LIN {X 0,Y 178.486,Z 136.368,A -85,B 0,C 180,E1 -22471.803,E2 -22471.803} C_VEL
LIN {X 0,Y 178.51,Z 136.363,A -85,B 0,C 180,E1 -22476.815,E2 -22476.815} C_VEL
LIN {X 0,Y 178.649,Z 136.34,A -85,B 0,C 180,E1 -22481.657,E2 -22481.657} C_VEL
LIN {X 0,Y 178.666,Z 136.339,A -85,B 0,C 180,E1 -22486.349,E2 -22486.349} C_VEL
LIN {X 0,Y 178.957,Z 136.319,A -85,B 0,C 180,E1 -22490.962,E2 -22490.962} C_VEL
LIN {X 0,Y 179.152,Z 136.294,A -85,B 0,C 180,E1 -22497.752,E2 -22497.752} C_VEL
LIN {X 0,Y 179.369,Z 136.252,A -85,B 0,C 180,E1 -22500,E2 -22500} C_VEL
LIN {X 0,Y 178.86,Z 136.321,A -85,B 0,C 180,E1 -22504.508,E2 -22504.508} C_VEL
LIN {X 0,Y 178.907,Z 136.301,A -85,B 0,C 180,E1 -22509.041,E2 -22509.041} C_VEL
LIN {X 0,Y 178.659,Z 136.355,A -85,B 0,C 180,E1 -22513.653,E2 -22513.653} C_VEL
LIN {X 0,Y 178.654,Z 136.338,A -85,B 0,C 180,E1 -22519.245,E2 -22519.245} C_VEL
LIN {X 0,Y 178.535,Z 136.348,A -85,B 0,C 180,E1 -22525.125,E2 -22525.125} C_VEL
LIN {X 0,Y 178.522,Z 136.362,A -85,B 0,C 180,E1 -22529.994,E2 -22529.994} C_VEL
LIN {X 0,Y 178.484,Z 136.378,A -85,B 0,C 180,E1 -22534.22,E2 -22534.22} C_VEL
LIN {X 0,Y 178.434,Z 136.535,A -85,B 0,C 180,E1 -22539.429,E2 -22539.429} C_VEL
LIN {X 0,Y 179.248,Z 138.944,A -85,B 0,C 180,E1 -22539.944,E2 -22539.944} C_VEL
LIN {X 0,Y 181.215,Z 141.18,A -85,B 0,C 180,E1 -22540.917,E2 -22540.917} C_VEL
LIN {X 0,Y 182.206,Z 142.05,A -85,B 0,C 180,E1 -22541.375,E2 -22541.375} C_VEL
LIN {X 0,Y 184.192,Z 145.249,A -85,B 0,C 180,E1 -22542.353,E2 -22542.353} C_VEL
LIN {X 0,Y 185.848,Z 147.075,A -85,B 0,C 180,E1 -22543.088,E2 -22543.088} C_VEL
LIN {X 0,Y 188.488,Z 150.745,A -85,B 0,C 180,E1 -22544.254,E2 -22544.254} C_VEL
LIN {X 0,Y 195.166,Z 160.483,A -85,B 0,C 180,E1 -22546.984,E2 -22546.984} C_VEL
LIN {X 0,Y 201.382,Z 170.518,A -85,B 0,C 180,E1 -22549.304,E2 -22549.304} C_VEL
LIN {X 0,Y 207.113,Z 180.976,A -85,B 0,C 180,E1 -22551.304,E2 -22551.304} C_VEL
LIN {X 0,Y 212.528,Z 194.015,A -85,B 0,C 180,E1 -22553.179,E2 -22553.179} C_VEL
LIN {X 0,Y 208.581,Z 264.938,A -85,B 0,C 180,E1 -22555.422,E2 -22555.422} C_VEL
LIN {X 0,Y 207.1,Z 278.824,A -85,B 0,C 180,E1 -22556.169,E2 -22556.169} C_VEL
LIN {X 0,Y 204.905,Z 292.956,A -85,B 0,C 180,E1 -22557.303,E2 -22557.303} C_VEL
LIN {X 0,Y 201.992,Z 306.924,A -85,B 0,C 180,E1 -22558.832,E2 -22558.832} C_VEL
LIN {X 0,Y 198.824,Z 319.397,A -85,B 0,C 180,E1 -22560.63,E2 -22560.63} C_VEL
LIN {X 0,Y 195.579,Z 330.767,A -85,B 0,C 180,E1 -22562.732,E2 -22562.732} C_VEL
LIN {X 0,Y 192.154,Z 341.225,A -85,B 0,C 180,E1 -22565.127,E2 -22565.127} C_VEL
LIN {X 0,Y 188.423,Z 351.62,A -85,B 0,C 180,E1 -22568.1,E2 -22568.1} C_VEL
LIN {X 0,Y 185.325,Z 360.19,A -85,B 0,C 180,E1 -22571.196,E2 -22571.196} C_VEL
LIN {X 0,Y 182.454,Z 367.978,A -85,B 0,C 180,E1 -22574.699,E2 -22574.699} C_VEL
LIN {X 0,Y 179.719,Z 375.042,A -85,B 0,C 180,E1 -22578.725,E2 -22578.725} C_VEL
LIN {X 0,Y 177.688,Z 380.92,A -85,B 0,C 180,E1 -22583.186,E2 -22583.186} C_VEL
LIN {X 0,Y 176.565,Z 385.24,A -85,B 0,C 180,E1 -22587.719,E2 -22587.719} C_VEL
LIN {X 0,Y 176.02,Z 388.135,A -85,B 0,C 180,E1 -22592.289,E2 -22592.289} C_VEL
LIN {X 0,Y 175.937,Z 389.074,A -85,B 0,C 180,E1 -22594.583,E2 -22594.583} C_VEL
LIN {X 0,Y 175.912,Z 389.967,A -85,B 0,C 180,E1 -22599.196,E2 -22599.196} C_VEL
LIN {X 0,Y 176.481,Z 389.534,A -85,B 0,C 180,E1 -22603.824,E2 -22603.824} C_VEL
LIN {X 0,Y 177.992,Z 387.659,A -85,B 0,C 180,E1 -22608.622,E2 -22608.622} C_VEL
LIN {X 0,Y 180.078,Z 384.585,A -85,B 0,C 180,E1 -22612.972,E2 -22612.972} C_VEL
LIN {X 0,Y 183.234,Z 379.874,A -85,B 0,C 180,E1 -22617.405,E2 -22617.405} C_VEL
LIN {X 0,Y 186.251,Z 375.283,A -85,B 0,C 180,E1 -22620.625,E2 -22620.625} C_VEL
LIN {X 0,Y 190.461,Z 368.593,A -85,B 0,C 180,E1 -22624.245,E2 -22624.245} C_VEL
LIN {X 0,Y 195.256,Z 360.22,A -85,B 0,C 180,E1 -22627.727,E2 -22627.727} C_VEL
LIN {X 0,Y 199.905,Z 351.456,A -85,B 0,C 180,E1 -22630.572,E2 -22630.572} C_VEL
LIN {X 0,Y 204.196,Z 342.773,A -85,B 0,C 180,E1 -22632.825,E2 -22632.825} C_VEL
LIN {X 0,Y 209.112,Z 331.656,A -85,B 0,C 180,E1 -22635.107,E2 -22635.107} C_VEL
LIN {X 0,Y 213.096,Z 321.091,A -85,B 0,C 180,E1 -22636.861,E2 -22636.861} C_VEL
LIN {X 0,Y 217.194,Z 308.734,A -85,B 0,C 180,E1 -22638.442,E2 -22638.442} C_VEL
LIN {X 0,Y 220.596,Z 296.079,A -85,B 0,C 180,E1 -22639.697,E2 -22639.697} C_VEL
LIN {X 0,Y 223.426,Z 281.915,A -85,B 0,C 180,E1 -22640.76,E2 -22640.76} C_VEL
LIN {X 0,Y 225.438,Z 268.079,A -85,B 0,C 180,E1 -22641.453,E2 -22641.453} C_VEL
LIN {X 0,Y 227.196,Z 245.698,A -85,B 0,C 180,E1 -22642.138,E2 -22642.138} C_VEL
LIN {X 0,Y 229.57,Z 209.78,A -85,B 0,C 180,E1 -22643.147,E2 -22643.147} C_VEL
LIN {X 0,Y 223.747,Z 197.099,A -85,B 0,C 180,E1 -22645.613,E2 -22645.613} C_VEL
LIN {X 0,Y 219.607,Z 189.431,A -85,B 0,C 180,E1 -22647.466,E2 -22647.466} C_VEL
LIN {X 0,Y 213.902,Z 180.454,A -85,B 0,C 180,E1 -22650.201,E2 -22650.201} C_VEL
LIN {X 0,Y 208.778,Z 173.011,A -85,B 0,C 180,E1 -22652.947,E2 -22652.947} C_VEL
LIN {X 0,Y 205.032,Z 168.032,A -85,B 0,C 180,E1 -22655.171,E2 -22655.171} C_VEL
LIN {X 0,Y 202.022,Z 163.972,A -85,B 0,C 180,E1 -22657.155,E2 -22657.155} C_VEL
LIN {X 0,Y 199.176,Z 160.496,A -85,B 0,C 180,E1 -22659.202,E2 -22659.202} C_VEL
LIN {X 0,Y 198.282,Z 159.146,A -85,B 0,C 180,E1 -22659.917,E2 -22659.917} C_VEL
LIN {X 0,Y 195.65,Z 156.447,A -85,B 0,C 180,E1 -22662.073,E2 -22662.073} C_VEL
LIN {X 0,Y 194.186,Z 153.936,A -85,B 0,C 180,E1 -22663.508,E2 -22663.508} C_VEL
LIN {X 0,Y 191.565,Z 151.793,A -85,B 0,C 180,E1 -22666.136,E2 -22666.136} C_VEL
LIN {X 0,Y 189.782,Z 148.386,A -85,B 0,C 180,E1 -22668.518,E2 -22668.518} C_VEL
LIN {X 0,Y 186.239,Z 145.756,A -85,B 0,C 180,E1 -22674.315,E2 -22674.315} C_VEL
LIN {X 0,Y 185.281,Z 143.481,A -85,B 0,C 180,E1 -22677.418,E2 -22677.418} C_VEL
LIN {X 0,Y 185.143,Z 142.415,A -85,B 0,C 180,E1 -22678.368,E2 -22678.368} C_VEL
LIN {X 0,Y 185.004,Z 142.485,A -85,B 0,C 180,E1 -22686.817,E2 -22686.817} C_VEL
LIN {X 0,Y 186.711,Z 146.523,A -85,B 0,C 180,E1 -22692.499,E2 -22692.499} C_VEL
LIN {X 0,Y 189.834,Z 148.662,A -85,B 0,C 180,E1 -22697.311,E2 -22697.311} C_VEL
LIN {X 0,Y 191.307,Z 151.577,A -85,B 0,C 180,E1 -22699.307,E2 -22699.307} C_VEL
LIN {X 0,Y 193.883,Z 153.809,A -85,B 0,C 180,E1 -22701.951,E2 -22701.951} C_VEL
LIN {X 0,Y 194.461,Z 154.358,A -85,B 0,C 180,E1 -22702.494,E2 -22702.494} C_VEL
LIN {X 0,Y 196.476,Z 157.499,A -85,B 0,C 180,E1 -22704.38,E2 -22704.38} C_VEL
LIN {X 0,Y 198.823,Z 159.877,A -85,B 0,C 180,E1 -22706.239,E2 -22706.239} C_VEL
LIN {X 0,Y 201.386,Z 163.367,A -85,B 0,C 180,E1 -22708.148,E2 -22708.148} C_VEL
LIN {X 0,Y 203.327,Z 165.931,A -85,B 0,C 180,E1 -22709.473,E2 -22709.473} C_VEL
LIN {X 0,Y 207.068,Z 171.804,A -85,B 0,C 180,E1 -22711.87,E2 -22711.87} C_VEL
LIN {X 0,Y 209.974,Z 176.459,A -85,B 0,C 180,E1 -22713.567,E2 -22713.567} C_VEL
LIN {X 0,Y 214.704,Z 184.513,A -85,B 0,C 180,E1 -22716.1,E2 -22716.1} C_VEL
LIN {X 0,Y 220.915,Z 196.355,A -85,B 0,C 180,E1 -22719.107,E2 -22719.107} C_VEL
LIN {X 0,Y 226.829,Z 209.325,A -85,B 0,C 180,E1 -22721.726,E2 -22721.726} C_VEL
LIN {X 0,Y 229.29,Z 215.482,A -85,B 0,C 180,E1 -22722.771,E2 -22722.771} C_VEL
LIN {X 0,Y 226.765,Z 253.212,A -85,B 0,C 180,E1 -22723.821,E2 -22723.821} C_VEL
LIN {X 0,Y 225.889,Z 259.067,A -85,B 0,C 180,E1 -22723.837,E2 -22723.837} C_VEL
LIN {X 0,Y 220.831,Z 276.116,A -85,B 0,C 180,E1 -22723.343,E2 -22723.343} C_VEL
LIN {X 0,Y 219.402,Z 281.85,A -85,B 0,C 180,E1 -22723.411,E2 -22723.411} C_VEL
LIN {X 0,Y 219.081,Z 283.768,A -85,B 0,C 180,E1 -22723.5,E2 -22723.5} C_VEL
LIN {X 0,Y 216.297,Z 297.815,A -85,B 0,C 180,E1 -22724.37,E2 -22724.37} C_VEL
LIN {X 0,Y 212.928,Z 310.546,A -85,B 0,C 180,E1 -22725.461,E2 -22725.461} C_VEL
LIN {X 0,Y 208.683,Z 323.745,A -85,B 0,C 180,E1 -22727.001,E2 -22727.001} C_VEL
LIN {X 0,Y 204.032,Z 335.665,A -85,B 0,C 180,E1 -22728.794,E2 -22728.794} C_VEL
LIN {X 0,Y 198.988,Z 347.089,A -85,B 0,C 180,E1 -22731.032,E2 -22731.032} C_VEL
LIN {X 0,Y 193.433,Z 358.123,A -85,B 0,C 180,E1 -22733.813,E2 -22733.813} C_VEL
LIN {X 0,Y 188.464,Z 366.89,A -85,B 0,C 180,E1 -22736.63,E2 -22736.63} C_VEL
LIN {X 0,Y 183.38,Z 375.311,A -85,B 0,C 180,E1 -22740.117,E2 -22740.117} C_VEL
LIN {X 0,Y 179.533,Z 381.206,A -85,B 0,C 180,E1 -22743.245,E2 -22743.245} C_VEL
LIN {X 0,Y 176.298,Z 386.092,A -85,B 0,C 180,E1 -22746.506,E2 -22746.506} C_VEL
LIN {X 0,Y 173.054,Z 391.158,A -85,B 0,C 180,E1 -22751.041,E2 -22751.041} C_VEL
LIN {X 0,Y 170.616,Z 394.743,A -85,B 0,C 180,E1 -22755.691,E2 -22755.691} C_VEL
LIN {X 0,Y 169.324,Z 396.953,A -85,B 0,C 180,E1 -22760.443,E2 -22760.443} C_VEL
LIN {X 0,Y 168.858,Z 397.835,A -85,B 0,C 180,E1 -22765.225,E2 -22765.225} C_VEL
LIN {X 0,Y 168.943,Z 397.392,A -85,B 0,C 180,E1 -22770,E2 -22770} C_VEL
LIN {X 0,Y 168.833,Z 396.62,A -85,B 0,C 180,E1 -22772.506,E2 -22772.506} C_VEL
LIN {X 0,Y 168.962,Z 394.168,A -85,B 0,C 180,E1 -22777.168,E2 -22777.168} C_VEL
LIN {X 0,Y 169.478,Z 391.316,A -85,B 0,C 180,E1 -22780.754,E2 -22780.754} C_VEL
LIN {X 0,Y 170.853,Z 386.202,A -85,B 0,C 180,E1 -22785.508,E2 -22785.508} C_VEL
LIN {X 0,Y 172.563,Z 381.246,A -85,B 0,C 180,E1 -22789.015,E2 -22789.015} C_VEL
LIN {X 0,Y 175.147,Z 374.083,A -85,B 0,C 180,E1 -22793.045,E2 -22793.045} C_VEL
LIN {X 0,Y 178.555,Z 365.268,A -85,B 0,C 180,E1 -22796.913,E2 -22796.913} C_VEL
LIN {X 0,Y 182.099,Z 356.008,A -85,B 0,C 180,E1 -22800.114,E2 -22800.114} C_VEL
LIN {X 0,Y 185.95,Z 345.785,A -85,B 0,C 180,E1 -22802.908,E2 -22802.908} C_VEL
LIN {X 0,Y 189.809,Z 334.101,A -85,B 0,C 180,E1 -22805.454,E2 -22805.454} C_VEL
LIN {X 0,Y 193.369,Z 322.05,A -85,B 0,C 180,E1 -22807.501,E2 -22807.501} C_VEL
LIN {X 0,Y 196.679,Z 309.03,A -85,B 0,C 180,E1 -22809.2,E2 -22809.2} C_VEL
LIN {X 0,Y 199.46,Z 295.554,A -85,B 0,C 180,E1 -22810.514,E2 -22810.514} C_VEL
LIN {X 0,Y 201.683,Z 280.974,A -85,B 0,C 180,E1 -22811.525,E2 -22811.525} C_VEL
LIN {X 0,Y 203.143,Z 266.315,A -85,B 0,C 180,E1 -22812.156,E2 -22812.156} C_VEL
LIN {X 0,Y 206.817,Z 201.907,A -85,B 0,C 180,E1 -22814.192,E2 -22814.192} C_VEL
LIN {X 0,Y 201.234,Z 187.244,A -85,B 0,C 180,E1 -22816.303,E2 -22816.303} C_VEL
LIN {X 0,Y 195.797,Z 175.404,A -85,B 0,C 180,E1 -22818.428,E2 -22818.428} C_VEL
LIN {X 0,Y 189.888,Z 163.919,A -85,B 0,C 180,E1 -22820.901,E2 -22820.901} C_VEL
LIN {X 0,Y 186.31,Z 158.007,A -85,B 0,C 180,E1 -22822.476,E2 -22822.476} C_VEL
LIN {X 0,Y 181.962,Z 151.818,A -85,B 0,C 180,E1 -22824.488,E2 -22824.488} C_VEL
LIN {X 0,Y 179.388,Z 148.301,A -85,B 0,C 180,E1 -22825.76,E2 -22825.76} C_VEL
LIN {X 0,Y 176.29,Z 144.63,A -85,B 0,C 180,E1 -22827.355,E2 -22827.355} C_VEL
LIN {X 0,Y 175.102,Z 142.606,A -85,B 0,C 180,E1 -22828.042,E2 -22828.042} C_VEL
LIN {X 0,Y 172.77,Z 140.563,A -85,B 0,C 180,E1 -22829.313,E2 -22829.313} C_VEL
LIN {X 0,Y 171.595,Z 137.936,A -85,B 0,C 180,E1 -22830.104,E2 -22830.104} C_VEL
LIN {X 0,Y 171.472,Z 137.24,A -85,B 0,C 180,E1 -22830.31,E2 -22830.31} C_VEL
LIN {X 0,Y 171.457,Z 137.238,A -85,B 0,C 180,E1 -22835.802,E2 -22835.802} C_VEL
LIN {X 0,Y 171.578,Z 137.22,A -85,B 0,C 180,E1 -22840.872,E2 -22840.872} C_VEL
LIN {X 0,Y 171.593,Z 137.225,A -85,B 0,C 180,E1 -22845.775,E2 -22845.775} C_VEL
LIN {X 0,Y 171.886,Z 137.199,A -85,B 0,C 180,E1 -22850.587,E2 -22850.587} C_VEL
LIN {X 0,Y 171.818,Z 137.189,A -85,B 0,C 180,E1 -22855.308,E2 -22855.308} C_VEL
LIN {X 0,Y 172.332,Z 137.127,A -85,B 0,C 180,E1 -22860,E2 -22860} C_VEL
LIN {X 0,Y 171.809,Z 137.201,A -85,B 0,C 180,E1 -22864.693,E2 -22864.693} C_VEL
LIN {X 0,Y 171.844,Z 137.177,A -85,B 0,C 180,E1 -22869.416,E2 -22869.416} C_VEL
LIN {X 0,Y 171.58,Z 137.237,A -85,B 0,C 180,E1 -22874.227,E2 -22874.227} C_VEL
LIN {X 0,Y 171.575,Z 137.222,A -85,B 0,C 180,E1 -22879.591,E2 -22879.591} C_VEL
LIN {X 0,Y 171.469,Z 137.228,A -85,B 0,C 180,E1 -22885.617,E2 -22885.617} C_VEL
LIN {X 0,Y 171.441,Z 137.239,A -85,B 0,C 180,E1 -22890.587,E2 -22890.587} C_VEL
LIN {X 0,Y 171.393,Z 137.302,A -85,B 0,C 180,E1 -22896.119,E2 -22896.119} C_VEL
LIN {X 0,Y 172.221,Z 139.853,A -85,B 0,C 180,E1 -22896.734,E2 -22896.734} C_VEL
LIN {X 0,Y 174.207,Z 142.08,A -85,B 0,C 180,E1 -22897.872,E2 -22897.872} C_VEL
LIN {X 0,Y 175.392,Z 143.049,A -85,B 0,C 180,E1 -22898.499,E2 -22898.499} C_VEL
LIN {X 0,Y 177.484,Z 146.372,A -85,B 0,C 180,E1 -22899.671,E2 -22899.671} C_VEL
LIN {X 0,Y 179.247,Z 148.253,A -85,B 0,C 180,E1 -22900.553,E2 -22900.553} C_VEL
LIN {X 0,Y 181.957,Z 151.964,A -85,B 0,C 180,E1 -22901.895,E2 -22901.895} C_VEL
LIN {X 0,Y 186.526,Z 158.471,A -85,B 0,C 180,E1 -22904.004,E2 -22904.004} C_VEL
LIN {X 0,Y 191.824,Z 166.326,A -85,B 0,C 180,E1 -22906.24,E2 -22906.24} C_VEL
LIN {X 0,Y 198.165,Z 176.886,A -85,B 0,C 180,E1 -22908.714,E2 -22908.714} C_VEL
LIN {X 0,Y 202.96,Z 185.998,A -85,B 0,C 180,E1 -22910.473,E2 -22910.473} C_VEL
LIN {X 0,Y 207.061,Z 196.134,A -85,B 0,C 180,E1 -22911.982,E2 -22911.982} C_VEL
LIN {X 0,Y 203.045,Z 264.915,A -85,B 0,C 180,E1 -22914.185,E2 -22914.185} C_VEL
LIN {X 0,Y 201.518,Z 278.875,A -85,B 0,C 180,E1 -22914.946,E2 -22914.946} C_VEL
LIN {X 0,Y 199.231,Z 293.039,A -85,B 0,C 180,E1 -22916.097,E2 -22916.097} C_VEL
LIN {X 0,Y 196.41,Z 306.148,A -85,B 0,C 180,E1 -22917.539,E2 -22917.539} C_VEL
LIN {X 0,Y 193.091,Z 318.804,A -85,B 0,C 180,E1 -22919.366,E2 -22919.366} C_VEL
LIN {X 0,Y 189.707,Z 330.306,A -85,B 0,C 180,E1 -22921.512,E2 -22921.512} C_VEL
LIN {X 0,Y 185.758,Z 341.839,A -85,B 0,C 180,E1 -22924.209,E2 -22924.209} C_VEL
LIN {X 0,Y 181.879,Z 352.16,A -85,B 0,C 180,E1 -22927.269,E2 -22927.269} C_VEL
LIN {X 0,Y 178.643,Z 360.666,A -85,B 0,C 180,E1 -22930.464,E2 -22930.464} C_VEL
LIN {X 0,Y 175.825,Z 367.743,A -85,B 0,C 180,E1 -22933.752,E2 -22933.752} C_VEL
LIN {X 0,Y 173.513,Z 373.633,A -85,B 0,C 180,E1 -22937.128,E2 -22937.128} C_VEL
LIN {X 0,Y 171.175,Z 379.925,A -85,B 0,C 180,E1 -22941.738,E2 -22941.738} C_VEL
LIN {X 0,Y 169.997,Z 383.551,A -85,B 0,C 180,E1 -22945.258,E2 -22945.258} C_VEL
LIN {X 0,Y 169.119,Z 387.107,A -85,B 0,C 180,E1 -22950,E2 -22950} C_VEL
LIN {X 0,Y 168.912,Z 388.672,A -85,B 0,C 180,E1 -22953.043,E2 -22953.043} C_VEL
LIN {X 0,Y 168.774,Z 389.877,A -85,B 0,C 180,E1 -22957.177,E2 -22957.177} C_VEL
LIN {X 0,Y 169.03,Z 390.073,A -85,B 0,C 180,E1 -22961.999,E2 -22961.999} C_VEL
LIN {X 0,Y 170.17,Z 388.934,A -85,B 0,C 180,E1 -22966.804,E2 -22966.804} C_VEL
LIN {X 0,Y 172.11,Z 386.428,A -85,B 0,C 180,E1 -22971.562,E2 -22971.562} C_VEL
LIN {X 0,Y 175.033,Z 382.448,A -85,B 0,C 180,E1 -22976.211,E2 -22976.211} C_VEL
LIN {X 0,Y 178.908,Z 376.877,A -85,B 0,C 180,E1 -22980.709,E2 -22980.709} C_VEL
LIN {X 0,Y 183.174,Z 370.555,A -85,B 0,C 180,E1 -22984.467,E2 -22984.467} C_VEL
LIN {X 0,Y 187.755,Z 363.199,A -85,B 0,C 180,E1 -22987.844,E2 -22987.844} C_VEL
LIN {X 0,Y 192.785,Z 354.366,A -85,B 0,C 180,E1 -22991.01,E2 -22991.01} C_VEL
LIN {X 0,Y 198.038,Z 344.351,A -85,B 0,C 180,E1 -22993.79,E2 -22993.79} C_VEL
LIN {X 0,Y 202.947,Z 334.007,A -85,B 0,C 180,E1 -22996.022,E2 -22996.022} C_VEL
LIN {X 0,Y 207.194,Z 323.327,A -85,B 0,C 180,E1 -22997.902,E2 -22997.902} C_VEL
LIN {X 0,Y 211.493,Z 311.505,A -85,B 0,C 180,E1 -22999.477,E2 -22999.477} C_VEL
LIN {X 0,Y 214.919,Z 299.537,A -85,B 0,C 180,E1 -23000.769,E2 -23000.769} C_VEL
LIN {X 0,Y 218.012,Z 285.863,A -85,B 0,C 180,E1 -23001.885,E2 -23001.885} C_VEL
LIN {X 0,Y 220.37,Z 271.605,A -85,B 0,C 180,E1 -23002.688,E2 -23002.688} C_VEL
LIN {X 0,Y 221.867,Z 256.171,A -85,B 0,C 180,E1 -23003.228,E2 -23003.228} C_VEL
LIN {X 0,Y 224.935,Z 212.537,A -85,B 0,C 180,E1 -23004.439,E2 -23004.439} C_VEL
LIN {X 0,Y 219.404,Z 200.419,A -85,B 0,C 180,E1 -23006.937,E2 -23006.937} C_VEL
LIN {X 0,Y 215.998,Z 194.049,A -85,B 0,C 180,E1 -23008.559,E2 -23008.559} C_VEL
LIN {X 0,Y 210.252,Z 184.968,A -85,B 0,C 180,E1 -23011.485,E2 -23011.485} C_VEL
LIN {X 0,Y 205.74,Z 178.356,A -85,B 0,C 180,E1 -23014.061,E2 -23014.061} C_VEL
LIN {X 0,Y 202.638,Z 174.042,A -85,B 0,C 180,E1 -23016.016,E2 -23016.016} C_VEL
LIN {X 0,Y 199.776,Z 170.125,A -85,B 0,C 180,E1 -23018,E2 -23018} C_VEL
LIN {X 0,Y 197.006,Z 166.47,A -85,B 0,C 180,E1 -23020.122,E2 -23020.122} C_VEL
LIN {X 0,Y 196.04,Z 165.384,A -85,B 0,C 180,E1 -23020.905,E2 -23020.905} C_VEL
LIN {X 0,Y 193.487,Z 162.209,A -85,B 0,C 180,E1 -23023.192,E2 -23023.192} C_VEL
LIN {X 0,Y 192.499,Z 160.599,A -85,B 0,C 180,E1 -23024.21,E2 -23024.21} C_VEL
LIN {X 0,Y 189.879,Z 158.11,A -85,B 0,C 180,E1 -23027.032,E2 -23027.032} C_VEL
LIN {X 0,Y 188.318,Z 155.191,A -85,B 0,C 180,E1 -23029.245,E2 -23029.245} C_VEL
LIN {X 0,Y 184.947,Z 152.273,A -85,B 0,C 180,E1 -23035.368,E2 -23035.368} C_VEL
LIN {X 0,Y 184.246,Z 149.993,A -85,B 0,C 180,E1 -23038.224,E2 -23038.224} C_VEL
LIN {X 0,Y 184.15,Z 149.427,A -85,B 0,C 180,E1 -23038.906,E2 -23038.906} C_VEL
LIN {X 0,Y 184.083,Z 149.537,A -85,B 0,C 180,E1 -23046.576,E2 -23046.576} C_VEL
LIN {X 0,Y 185.721,Z 153.53,A -85,B 0,C 180,E1 -23052.287,E2 -23052.287} C_VEL
LIN {X 0,Y 188.478,Z 155.492,A -85,B 0,C 180,E1 -23056.727,E2 -23056.727} C_VEL
LIN {X 0,Y 190.072,Z 158.501,A -85,B 0,C 180,E1 -23058.951,E2 -23058.951} C_VEL
LIN {X 0,Y 192.868,Z 161.11,A -85,B 0,C 180,E1 -23061.896,E2 -23061.896} C_VEL
LIN {X 0,Y 195.276,Z 164.638,A -85,B 0,C 180,E1 -23064.191,E2 -23064.191} C_VEL
LIN {X 0,Y 197.012,Z 166.46,A -85,B 0,C 180,E1 -23065.61,E2 -23065.61} C_VEL
LIN {X 0,Y 200.96,Z 171.847,A -85,B 0,C 180,E1 -23068.581,E2 -23068.581} C_VEL
LIN {X 0,Y 205.164,Z 178.66,A -85,B 0,C 180,E1 -23071.397,E2 -23071.397} C_VEL
LIN {X 0,Y 209.109,Z 185.297,A -85,B 0,C 180,E1 -23073.75,E2 -23073.75} C_VEL
LIN {X 0,Y 214.505,Z 195.407,A -85,B 0,C 180,E1 -23076.665,E2 -23076.665} C_VEL
LIN {X 0,Y 219.297,Z 205.378,A -85,B 0,C 180,E1 -23079.022,E2 -23079.022} C_VEL
LIN {X 0,Y 223.957,Z 216.249,A -85,B 0,C 180,E1 -23081.163,E2 -23081.163} C_VEL
LIN {X 0,Y 224.59,Z 217.837,A -85,B 0,C 180,E1 -23081.445,E2 -23081.445} C_VEL
LIN {X 0,Y 220.71,Z 272.075,A -85,B 0,C 180,E1 -23082.997,E2 -23082.997} C_VEL
LIN {X 0,Y 219.081,Z 283.768,A -85,B 0,C 180,E1 -23083.5,E2 -23083.5} C_VEL
LIN {X 0,Y 217.68,Z 289.476,A -85,B 0,C 180,E1 -23083.681,E2 -23083.681} C_VEL
LIN {X 0,Y 213.779,Z 298.62,A -85,B 0,C 180,E1 -23083.711,E2 -23083.711} C_VEL
LIN {X 0,Y 209.463,Z 307.524,A -85,B 0,C 180,E1 -23083.88,E2 -23083.88} C_VEL
LIN {X 0,Y 207.419,Z 312.852,A -85,B 0,C 180,E1 -23084.29,E2 -23084.29} C_VEL
LIN {X 0,Y 202.99,Z 325.564,A -85,B 0,C 180,E1 -23085.831,E2 -23085.831} C_VEL
LIN {X 0,Y 198.232,Z 337.132,A -85,B 0,C 180,E1 -23087.653,E2 -23087.653} C_VEL
LIN {X 0,Y 192.771,Z 348.823,A -85,B 0,C 180,E1 -23090.054,E2 -23090.054} C_VEL
LIN {X 0,Y 187.755,Z 358.279,A -85,B 0,C 180,E1 -23092.535,E2 -23092.535} C_VEL
LIN {X 0,Y 182.55,Z 366.993,A -85,B 0,C 180,E1 -23095.399,E2 -23095.399} C_VEL
LIN {X 0,Y 177.222,Z 375.368,A -85,B 0,C 180,E1 -23098.967,E2 -23098.967} C_VEL
LIN {X 0,Y 173.203,Z 381.22,A -85,B 0,C 180,E1 -23102.184,E2 -23102.184} C_VEL
LIN {X 0,Y 169.592,Z 386.311,A -85,B 0,C 180,E1 -23105.74,E2 -23105.74} C_VEL
LIN {X 0,Y 166.295,Z 391.098,A -85,B 0,C 180,E1 -23110.239,E2 -23110.239} C_VEL
LIN {X 0,Y 163.7,Z 394.649,A -85,B 0,C 180,E1 -23115.072,E2 -23115.072} C_VEL
LIN {X 0,Y 162.311,Z 396.828,A -85,B 0,C 180,E1 -23120.026,E2 -23120.026} C_VEL
LIN {X 0,Y 161.76,Z 397.679,A -85,B 0,C 180,E1 -23125.015,E2 -23125.015} C_VEL
LIN {X 0,Y 161.761,Z 397.591,A -85,B 0,C 180,E1 -23127.817,E2 -23127.817} C_VEL
LIN {X 0,Y 161.842,Z 397.206,A -85,B 0,C 180,E1 -23130,E2 -23130} C_VEL
LIN {X 0,Y 161.756,Z 396.46,A -85,B 0,C 180,E1 -23132.49,E2 -23132.49} C_VEL
LIN {X 0,Y 161.905,Z 393.932,A -85,B 0,C 180,E1 -23137.482,E2 -23137.482} C_VEL
LIN {X 0,Y 162.742,Z 389.93,A -85,B 0,C 180,E1 -23142.469,E2 -23142.469} C_VEL
LIN {X 0,Y 164.543,Z 384.342,A -85,B 0,C 180,E1 -23147.396,E2 -23147.396} C_VEL
LIN {X 0,Y 166.893,Z 378.022,A -85,B 0,C 180,E1 -23151.621,E2 -23151.621} C_VEL
LIN {X 0,Y 170.036,Z 370.14,A -85,B 0,C 180,E1 -23155.721,E2 -23155.721} C_VEL
LIN {X 0,Y 173.395,Z 361.9,A -85,B 0,C 180,E1 -23159.103,E2 -23159.103} C_VEL
LIN {X 0,Y 177.421,Z 351.972,A -85,B 0,C 180,E1 -23162.327,E2 -23162.327} C_VEL
LIN {X 0,Y 181.523,Z 340.924,A -85,B 0,C 180,E1 -23165.163,E2 -23165.163} C_VEL
LIN {X 0,Y 185.554,Z 328.619,A -85,B 0,C 180,E1 -23167.643,E2 -23167.643} C_VEL
LIN {X 0,Y 189.098,Z 316.411,A -85,B 0,C 180,E1 -23169.528,E2 -23169.528} C_VEL
LIN {X 0,Y 192.391,Z 302.85,A -85,B 0,C 180,E1 -23171.112,E2 -23171.112} C_VEL
LIN {X 0,Y 195.077,Z 288.65,A -85,B 0,C 180,E1 -23172.318,E2 -23172.318} C_VEL
LIN {X 0,Y 197.02,Z 273.931,A -85,B 0,C 180,E1 -23173.163,E2 -23173.163} C_VEL
LIN {X 0,Y 198.847,Z 247.466,A -85,B 0,C 180,E1 -23174.059,E2 -23174.059} C_VEL
LIN {X 0,Y 201.431,Z 203.981,A -85,B 0,C 180,E1 -23175.451,E2 -23175.451} C_VEL
LIN {X 0,Y 195.716,Z 188.866,A -85,B 0,C 180,E1 -23177.765,E2 -23177.765} C_VEL
LIN {X 0,Y 189.867,Z 176.201,A -85,B 0,C 180,E1 -23180.233,E2 -23180.233} C_VEL
LIN {X 0,Y 183.905,Z 164.91,A -85,B 0,C 180,E1 -23182.948,E2 -23182.948} C_VEL
LIN {X 0,Y 178.64,Z 157.349,A -85,B 0,C 180,E1 -23185.486,E2 -23185.486} C_VEL
LIN {X 0,Y 175.577,Z 153.226,A -85,B 0,C 180,E1 -23187.088,E2 -23187.088} C_VEL
LIN {X 0,Y 173,Z 149.834,A -85,B 0,C 180,E1 -23188.527,E2 -23188.527} C_VEL
LIN {X 0,Y 172.172,Z 148.661,A -85,B 0,C 180,E1 -23189.016,E2 -23189.016} C_VEL
LIN {X 0,Y 169.628,Z 145.845,A -85,B 0,C 180,E1 -23190.528,E2 -23190.528} C_VEL
LIN {X 0,Y 168.455,Z 143.707,A -85,B 0,C 180,E1 -23191.329,E2 -23191.329} C_VEL
LIN {X 0,Y 166.023,Z 141.89,A -85,B 0,C 180,E1 -23192.865,E2 -23192.865} C_VEL
LIN {X 0,Y 164.703,Z 139.463,A -85,B 0,C 180,E1 -23193.875,E2 -23193.875} C_VEL
LIN {X 0,Y 164.433,Z 138.119,A -85,B 0,C 180,E1 -23194.259,E2 -23194.259} C_VEL
LIN {X 0,Y 164.484,Z 138.108,A -85,B 0,C 180,E1 -23200.051,E2 -23200.051} C_VEL
LIN {X 0,Y 164.542,Z 138.11,A -85,B 0,C 180,E1 -23205.151,E2 -23205.151} C_VEL
LIN {X 0,Y 164.801,Z 138.08,A -85,B 0,C 180,E1 -23210.179,E2 -23210.179} C_VEL
LIN {X 0,Y 164.848,Z 138.062,A -85,B 0,C 180,E1 -23212.652,E2 -23212.652} C_VEL
LIN {X 0,Y 165.048,Z 138.051,A -85,B 0,C 180,E1 -23217.56,E2 -23217.56} C_VEL
LIN {X 0,Y 165.294,Z 138.002,A -85,B 0,C 180,E1 -23220,E2 -23220} C_VEL
LIN {X 0,Y 164.757,Z 138.08,A -85,B 0,C 180,E1 -23224.894,E2 -23224.894} C_VEL
LIN {X 0,Y 164.825,Z 138.07,A -85,B 0,C 180,E1 -23227.35,E2 -23227.35} C_VEL
LIN {X 0,Y 164.702,Z 138.068,A -85,B 0,C 180,E1 -23231.061,E2 -23231.061} C_VEL
LIN {X 0,Y 164.503,Z 138.092,A -85,B 0,C 180,E1 -23237.402,E2 -23237.402} C_VEL
LIN {X 0,Y 164.52,Z 138.105,A -85,B 0,C 180,E1 -23239.984,E2 -23239.984} C_VEL
LIN {X 0,Y 164.394,Z 138.111,A -85,B 0,C 180,E1 -23246.135,E2 -23246.135} C_VEL
LIN {X 0,Y 164.394,Z 138.247,A -85,B 0,C 180,E1 -23252.199,E2 -23252.199} C_VEL
LIN {X 0,Y 165.252,Z 140.842,A -85,B 0,C 180,E1 -23252.958,E2 -23252.958} C_VEL
LIN {X 0,Y 167.27,Z 143.042,A -85,B 0,C 180,E1 -23254.331,E2 -23254.331} C_VEL
LIN {X 0,Y 168.599,Z 143.93,A -85,B 0,C 180,E1 -23255.144,E2 -23255.144} C_VEL
LIN {X 0,Y 170.318,Z 146.916,A -85,B 0,C 180,E1 -23256.291,E2 -23256.291} C_VEL
LIN {X 0,Y 172.64,Z 149.319,A -85,B 0,C 180,E1 -23257.636,E2 -23257.636} C_VEL
LIN {X 0,Y 175.288,Z 152.993,A -85,B 0,C 180,E1 -23259.14,E2 -23259.14} C_VEL
LIN {X 0,Y 176.681,Z 154.864,A -85,B 0,C 180,E1 -23259.887,E2 -23259.887} C_VEL
LIN {X 0,Y 180.01,Z 159.435,A -85,B 0,C 180,E1 -23261.585,E2 -23261.585} C_VEL
LIN {X 0,Y 185.561,Z 167.501,A -85,B 0,C 180,E1 -23264.182,E2 -23264.182} C_VEL
LIN {X 0,Y 191.821,Z 177.649,A -85,B 0,C 180,E1 -23266.848,E2 -23266.848} C_VEL
LIN {X 0,Y 198.206,Z 189.59,A -85,B 0,C 180,E1 -23269.358,E2 -23269.358} C_VEL
LIN {X 0,Y 201.692,Z 198.33,A -85,B 0,C 180,E1 -23270.725,E2 -23270.725} C_VEL
LIN {X 0,Y 197.456,Z 266.085,A -85,B 0,C 180,E1 -23272.926,E2 -23272.926} C_VEL
LIN {X 0,Y 195.796,Z 280.424,A -85,B 0,C 180,E1 -23273.763,E2 -23273.763} C_VEL
LIN {X 0,Y 193.431,Z 294.228,A -85,B 0,C 180,E1 -23274.934,E2 -23274.934} C_VEL
LIN {X 0,Y 190.49,Z 307.117,A -85,B 0,C 180,E1 -23276.399,E2 -23276.399} C_VEL
LIN {X 0,Y 187.056,Z 319.617,A -85,B 0,C 180,E1 -23278.265,E2 -23278.265} C_VEL
LIN {X 0,Y 183.521,Z 331.006,A -85,B 0,C 180,E1 -23280.459,E2 -23280.459} C_VEL
LIN {X 0,Y 179.42,Z 342.45,A -85,B 0,C 180,E1 -23283.227,E2 -23283.227} C_VEL
LIN {X 0,Y 175.388,Z 352.686,A -85,B 0,C 180,E1 -23286.378,E2 -23286.378} C_VEL
LIN {X 0,Y 171.995,Z 361.135,A -85,B 0,C 180,E1 -23289.677,E2 -23289.677} C_VEL
LIN {X 0,Y 168.6,Z 369.22,A -85,B 0,C 180,E1 -23293.659,E2 -23293.659} C_VEL
LIN {X 0,Y 165.852,Z 375.741,A -85,B 0,C 180,E1 -23297.768,E2 -23297.768} C_VEL
LIN {X 0,Y 163.639,Z 381.533,A -85,B 0,C 180,E1 -23302.598,E2 -23302.598} C_VEL
LIN {X 0,Y 162.395,Z 385.772,A -85,B 0,C 180,E1 -23307.52,E2 -23307.52} C_VEL
LIN {X 0,Y 161.835,Z 388.717,A -85,B 0,C 180,E1 -23312.769,E2 -23312.769} C_VEL
LIN {X 0,Y 161.679,Z 390.069,A -85,B 0,C 180,E1 -23317.493,E2 -23317.493} C_VEL
LIN {X 0,Y 162.001,Z 390.229,A -85,B 0,C 180,E1 -23322.528,E2 -23322.528} C_VEL
LIN {X 0,Y 163.286,Z 389.051,A -85,B 0,C 180,E1 -23327.535,E2 -23327.535} C_VEL
LIN {X 0,Y 165.404,Z 386.495,A -85,B 0,C 180,E1 -23332.483,E2 -23332.483} C_VEL
LIN {X 0,Y 168.553,Z 382.468,A -85,B 0,C 180,E1 -23337.301,E2 -23337.301} C_VEL
LIN {X 0,Y 172.736,Z 376.854,A -85,B 0,C 180,E1 -23341.933,E2 -23341.933} C_VEL
LIN {X 0,Y 177.244,Z 370.485,A -85,B 0,C 180,E1 -23345.794,E2 -23345.794} C_VEL
LIN {X 0,Y 182.367,Z 362.62,A -85,B 0,C 180,E1 -23349.434,E2 -23349.434} C_VEL
LIN {X 0,Y 187.393,Z 354.185,A -85,B 0,C 180,E1 -23352.46,E2 -23352.46} C_VEL
LIN {X 0,Y 192.911,Z 344.101,A -85,B 0,C 180,E1 -23355.269,E2 -23355.269} C_VEL
LIN {X 0,Y 198.362,Z 332.855,A -85,B 0,C 180,E1 -23357.687,E2 -23357.687} C_VEL
LIN {X 0,Y 203.012,Z 321.536,A -85,B 0,C 180,E1 -23359.607,E2 -23359.607} C_VEL
LIN {X 0,Y 207.394,Z 309.207,A -85,B 0,C 180,E1 -23361.206,E2 -23361.206} C_VEL
LIN {X 0,Y 211.035,Z 296.595,A -85,B 0,C 180,E1 -23362.469,E2 -23362.469} C_VEL
LIN {X 0,Y 214.047,Z 282.4,A -85,B 0,C 180,E1 -23363.557,E2 -23363.557} C_VEL
LIN {X 0,Y 216.292,Z 268.152,A -85,B 0,C 180,E1 -23364.259,E2 -23364.259} C_VEL
LIN {X 0,Y 218.211,Z 245.091,A -85,B 0,C 180,E1 -23364.967,E2 -23364.967} C_VEL
LIN {X 0,Y 220.404,Z 215.313,A -85,B 0,C 180,E1 -23365.79,E2 -23365.79} C_VEL
LIN {X 0,Y 215.532,Z 204.477,A -85,B 0,C 180,E1 -23368.14,E2 -23368.14} C_VEL
LIN {X 0,Y 212.34,Z 198.482,A -85,B 0,C 180,E1 -23369.754,E2 -23369.754} C_VEL
LIN {X 0,Y 206.325,Z 188.743,A -85,B 0,C 180,E1 -23373.051,E2 -23373.051} C_VEL
LIN {X 0,Y 200.866,Z 180.758,A -85,B 0,C 180,E1 -23376.494,E2 -23376.494} C_VEL
LIN {X 0,Y 197.7,Z 176.45,A -85,B 0,C 180,E1 -23378.767,E2 -23378.767} C_VEL
LIN {X 0,Y 194.518,Z 172.113,A -85,B 0,C 180,E1 -23381.367,E2 -23381.367} C_VEL
LIN {X 0,Y 191.881,Z 168.834,A -85,B 0,C 180,E1 -23383.816,E2 -23383.816} C_VEL
LIN {X 0,Y 191.098,Z 167.399,A -85,B 0,C 180,E1 -23384.672,E2 -23384.672} C_VEL
LIN {X 0,Y 188.508,Z 164.832,A -85,B 0,C 180,E1 -23387.587,E2 -23387.587} C_VEL
LIN {X 0,Y 187.059,Z 162.086,A -85,B 0,C 180,E1 -23389.74,E2 -23389.74} C_VEL
LIN {X 0,Y 183.919,Z 159.168,A -85,B 0,C 180,E1 -23395.788,E2 -23395.788} C_VEL
LIN {X 0,Y 183.268,Z 156.838,A -85,B 0,C 180,E1 -23398.764,E2 -23398.764} C_VEL
LIN {X 0,Y 183.173,Z 156.433,A -85,B 0,C 180,E1 -23399.45,E2 -23399.45} C_VEL
LIN {X 0,Y 183.198,Z 156.769,A -85,B 0,C 180,E1 -23406.608,E2 -23406.608} C_VEL
LIN {X 0,Y 184.555,Z 160.314,A -85,B 0,C 180,E1 -23411.67,E2 -23411.67} C_VEL
LIN {X 0,Y 187.232,Z 162.509,A -85,B 0,C 180,E1 -23416.281,E2 -23416.281} C_VEL
LIN {X 0,Y 189.09,Z 165.719,A -85,B 0,C 180,E1 -23418.89,E2 -23418.89} C_VEL
LIN {X 0,Y 191.346,Z 167.895,A -85,B 0,C 180,E1 -23421.336,E2 -23421.336} C_VEL
LIN {X 0,Y 193.909,Z 171.545,A -85,B 0,C 180,E1 -23423.845,E2 -23423.845} C_VEL
LIN {X 0,Y 195.163,Z 172.93,A -85,B 0,C 180,E1 -23424.914,E2 -23424.914} C_VEL
LIN {X 0,Y 198.847,Z 178.106,A -85,B 0,C 180,E1 -23427.823,E2 -23427.823} C_VEL
LIN {X 0,Y 203.149,Z 185.296,A -85,B 0,C 180,E1 -23430.833,E2 -23430.833} C_VEL
LIN {X 0,Y 207.828,Z 193.782,A -85,B 0,C 180,E1 -23433.721,E2 -23433.721} C_VEL
LIN {X 0,Y 212.376,Z 202.737,A -85,B 0,C 180,E1 -23436.245,E2 -23436.245} C_VEL
LIN {X 0,Y 216.904,Z 212.769,A -85,B 0,C 180,E1 -23438.566,E2 -23438.566} C_VEL
LIN {X 0,Y 220.02,Z 220.39,A -85,B 0,C 180,E1 -23440.076,E2 -23440.076} C_VEL
LIN {X 0,Y 216.118,Z 272.576,A -85,B 0,C 180,E1 -23441.587,E2 -23441.587} C_VEL
LIN {X 0,Y 213.919,Z 286.991,A -85,B 0,C 180,E1 -23442.249,E2 -23442.249} C_VEL
LIN {X 0,Y 210.853,Z 300.839,A -85,B 0,C 180,E1 -23443.187,E2 -23443.187} C_VEL
LIN {X 0,Y 207.419,Z 312.852,A -85,B 0,C 180,E1 -23444.29,E2 -23444.29} C_VEL
LIN {X 0,Y 205.262,Z 318.185,A -85,B 0,C 180,E1 -23444.758,E2 -23444.758} C_VEL
LIN {X 0,Y 200.196,Z 326.551,A -85,B 0,C 180,E1 -23445.247,E2 -23445.247} C_VEL
LIN {X 0,Y 194.839,Z 334.582,A -85,B 0,C 180,E1 -23445.875,E2 -23445.875} C_VEL
LIN {X 0,Y 192.246,Z 339.238,A -85,B 0,C 180,E1 -23446.57,E2 -23446.57} C_VEL
LIN {X 0,Y 186.714,Z 350.322,A -85,B 0,C 180,E1 -23448.967,E2 -23448.967} C_VEL
LIN {X 0,Y 181.244,Z 360.001,A -85,B 0,C 180,E1 -23451.653,E2 -23451.653} C_VEL
LIN {X 0,Y 175.913,Z 368.406,A -85,B 0,C 180,E1 -23454.598,E2 -23454.598} C_VEL
LIN {X 0,Y 170.419,Z 376.448,A -85,B 0,C 180,E1 -23458.277,E2 -23458.277} C_VEL
LIN {X 0,Y 165.642,Z 382.948,A -85,B 0,C 180,E1 -23462.178,E2 -23462.178} C_VEL
LIN {X 0,Y 162.403,Z 387.278,A -85,B 0,C 180,E1 -23465.54,E2 -23465.54} C_VEL
LIN {X 0,Y 159.576,Z 391.038,A -85,B 0,C 180,E1 -23469.369,E2 -23469.369} C_VEL
LIN {X 0,Y 156.807,Z 394.557,A -85,B 0,C 180,E1 -23474.4,E2 -23474.4} C_VEL
LIN {X 0,Y 155.282,Z 396.704,A -85,B 0,C 180,E1 -23479.569,E2 -23479.569} C_VEL
LIN {X 0,Y 154.687,Z 397.524,A -85,B 0,C 180,E1 -23484.786,E2 -23484.786} C_VEL
LIN {X 0,Y 154.744,Z 397.02,A -85,B 0,C 180,E1 -23490,E2 -23490} C_VEL
LIN {X 0,Y 154.663,Z 396.258,A -85,B 0,C 180,E1 -23492.604,E2 -23492.604} C_VEL
LIN {X 0,Y 154.843,Z 393.69,A -85,B 0,C 180,E1 -23497.825,E2 -23497.825} C_VEL
LIN {X 0,Y 155.777,Z 389.645,A -85,B 0,C 180,E1 -23503.036,E2 -23503.036} C_VEL
LIN {X 0,Y 157.739,Z 384.019,A -85,B 0,C 180,E1 -23508.172,E2 -23508.172} C_VEL
LIN {X 0,Y 160.338,Z 377.303,A -85,B 0,C 180,E1 -23512.787,E2 -23512.787} C_VEL
LIN {X 0,Y 163.611,Z 369.731,A -85,B 0,C 180,E1 -23516.809,E2 -23516.809} C_VEL
LIN {X 0,Y 167.166,Z 361.441,A -85,B 0,C 180,E1 -23520.298,E2 -23520.298} C_VEL
LIN {X 0,Y 171.406,Z 351.454,A -85,B 0,C 180,E1 -23523.609,E2 -23523.609} C_VEL
LIN {X 0,Y 175.739,Z 340.338,A -85,B 0,C 180,E1 -23526.503,E2 -23526.503} C_VEL
LIN {X 0,Y 179.94,Z 327.893,A -85,B 0,C 180,E1 -23529.035,E2 -23529.035} C_VEL
LIN {X 0,Y 183.633,Z 315.545,A -85,B 0,C 180,E1 -23530.95,E2 -23530.95} C_VEL
LIN {X 0,Y 187.093,Z 301.796,A -85,B 0,C 180,E1 -23532.543,E2 -23532.543} C_VEL
LIN {X 0,Y 189.853,Z 287.279,A -85,B 0,C 180,E1 -23533.77,E2 -23533.77} C_VEL
LIN {X 0,Y 191.773,Z 272.771,A -85,B 0,C 180,E1 -23534.586,E2 -23534.586} C_VEL
LIN {X 0,Y 194.407,Z 232.963,A -85,B 0,C 180,E1 -23535.925,E2 -23535.925} C_VEL
LIN {X 0,Y 196.121,Z 205.842,A -85,B 0,C 180,E1 -23536.796,E2 -23536.796} C_VEL
LIN {X 0,Y 190.687,Z 191.556,A -85,B 0,C 180,E1 -23539.142,E2 -23539.142} C_VEL
LIN {X 0,Y 184.877,Z 178.846,A -85,B 0,C 180,E1 -23541.779,E2 -23541.779} C_VEL
LIN {X 0,Y 179.648,Z 169.08,A -85,B 0,C 180,E1 -23544.328,E2 -23544.328} C_VEL
LIN {X 0,Y 174.866,Z 162.162,A -85,B 0,C 180,E1 -23546.798,E2 -23546.798} C_VEL
LIN {X 0,Y 172.295,Z 158.656,A -85,B 0,C 180,E1 -23548.232,E2 -23548.232} C_VEL
LIN {X 0,Y 169.293,Z 154.544,A -85,B 0,C 180,E1 -23550.036,E2 -23550.036} C_VEL
LIN {X 0,Y 166.707,Z 151.347,A -85,B 0,C 180,E1 -23551.688,E2 -23551.688} C_VEL
LIN {X 0,Y 165.747,Z 149.945,A -85,B 0,C 180,E1 -23552.353,E2 -23552.353} C_VEL
LIN {X 0,Y 163.369,Z 147.667,A -85,B 0,C 180,E1 -23553.988,E2 -23553.988} C_VEL
LIN {X 0,Y 161.786,Z 144.73,A -85,B 0,C 180,E1 -23555.285,E2 -23555.285} C_VEL
LIN {X 0,Y 159.205,Z 142.993,A -85,B 0,C 180,E1 -23557.278,E2 -23557.278} C_VEL
LIN {X 0,Y 157.784,Z 140.705,A -85,B 0,C 180,E1 -23558.612,E2 -23558.612} C_VEL
LIN {X 0,Y 157.36,Z 139.003,A -85,B 0,C 180,E1 -23559.178,E2 -23559.178} C_VEL
LIN {X 0,Y 157.47,Z 138.996,A -85,B 0,C 180,E1 -23564.468,E2 -23564.468} C_VEL
LIN {X 0,Y 157.725,Z 138.955,A -85,B 0,C 180,E1 -23569.733,E2 -23569.733} C_VEL
LIN {X 0,Y 157.805,Z 138.942,A -85,B 0,C 180,E1 -23572.322,E2 -23572.322} C_VEL
LIN {X 0,Y 158.256,Z 138.877,A -85,B 0,C 180,E1 -23580,E2 -23580} C_VEL
LIN {X 0,Y 157.763,Z 138.944,A -85,B 0,C 180,E1 -23587.681,E2 -23587.681} C_VEL
LIN {X 0,Y 157.636,Z 138.948,A -85,B 0,C 180,E1 -23591.237,E2 -23591.237} C_VEL
LIN {X 0,Y 157.463,Z 138.982,A -85,B 0,C 180,E1 -23595.534,E2 -23595.534} C_VEL
LIN {X 0,Y 157.416,Z 139,A -85,B 0,C 180,E1 -23600.927,E2 -23600.927} C_VEL
LIN {X 0,Y 157.3,Z 139.01,A -85,B 0,C 180,E1 -23607.183,E2 -23607.183} C_VEL
LIN {X 0,Y 158.022,Z 141.345,A -85,B 0,C 180,E1 -23608.018,E2 -23608.018} C_VEL
LIN {X 0,Y 159.86,Z 143.647,A -85,B 0,C 180,E1 -23609.643,E2 -23609.643} C_VEL
LIN {X 0,Y 161.935,Z 145.006,A -85,B 0,C 180,E1 -23611.215,E2 -23611.215} C_VEL
LIN {X 0,Y 163.606,Z 148.032,A -85,B 0,C 180,E1 -23612.569,E2 -23612.569} C_VEL
LIN {X 0,Y 166.137,Z 150.421,A -85,B 0,C 180,E1 -23614.288,E2 -23614.288} C_VEL
LIN {X 0,Y 168.441,Z 153.818,A -85,B 0,C 180,E1 -23615.834,E2 -23615.834} C_VEL
LIN {X 0,Y 170.1,Z 155.673,A -85,B 0,C 180,E1 -23616.84,E2 -23616.84} C_VEL
LIN {X 0,Y 173.83,Z 160.875,A -85,B 0,C 180,E1 -23619.019,E2 -23619.019} C_VEL
LIN {X 0,Y 177.15,Z 165.546,A -85,B 0,C 180,E1 -23620.796,E2 -23620.796} C_VEL
LIN {X 0,Y 182.582,Z 173.618,A -85,B 0,C 180,E1 -23623.455,E2 -23623.455} C_VEL
LIN {X 0,Y 188.576,Z 183.742,A -85,B 0,C 180,E1 -23626.134,E2 -23626.134} C_VEL
LIN {X 0,Y 193.915,Z 194.114,A -85,B 0,C 180,E1 -23628.351,E2 -23628.351} C_VEL
LIN {X 0,Y 196.385,Z 200.483,A -85,B 0,C 180,E1 -23629.388,E2 -23629.388} C_VEL
LIN {X 0,Y 192.123,Z 266.063,A -85,B 0,C 180,E1 -23631.548,E2 -23631.548} C_VEL
LIN {X 0,Y 190.395,Z 280.463,A -85,B 0,C 180,E1 -23632.396,E2 -23632.396} C_VEL
LIN {X 0,Y 187.936,Z 294.299,A -85,B 0,C 180,E1 -23633.584,E2 -23633.584} C_VEL
LIN {X 0,Y 184.653,Z 308.085,A -85,B 0,C 180,E1 -23635.187,E2 -23635.187} C_VEL
LIN {X 0,Y 181.094,Z 320.429,A -85,B 0,C 180,E1 -23637.091,E2 -23637.091} C_VEL
LIN {X 0,Y 177.012,Z 332.866,A -85,B 0,C 180,E1 -23639.588,E2 -23639.588} C_VEL
LIN {X 0,Y 173.145,Z 343.056,A -85,B 0,C 180,E1 -23642.175,E2 -23642.175} C_VEL
LIN {X 0,Y 168.932,Z 353.195,A -85,B 0,C 180,E1 -23645.417,E2 -23645.417} C_VEL
LIN {X 0,Y 165.381,Z 361.588,A -85,B 0,C 180,E1 -23648.826,E2 -23648.826} C_VEL
LIN {X 0,Y 161.825,Z 369.612,A -85,B 0,C 180,E1 -23652.954,E2 -23652.954} C_VEL
LIN {X 0,Y 158.931,Z 376.088,A -85,B 0,C 180,E1 -23657.227,E2 -23657.227} C_VEL
LIN {X 0,Y 156.625,Z 381.837,A -85,B 0,C 180,E1 -23662.264,E2 -23662.264} C_VEL
LIN {X 0,Y 155.304,Z 386.038,A -85,B 0,C 180,E1 -23667.407,E2 -23667.407} C_VEL
LIN {X 0,Y 154.741,Z 388.818,A -85,B 0,C 180,E1 -23672.604,E2 -23672.604} C_VEL
LIN {X 0,Y 154.626,Z 389.704,A -85,B 0,C 180,E1 -23675.216,E2 -23675.216} C_VEL
LIN {X 0,Y 154.7,Z 390.488,A -85,B 0,C 180,E1 -23680.47,E2 -23680.47} C_VEL
LIN {X 0,Y 155.6,Z 389.944,A -85,B 0,C 180,E1 -23685.724,E2 -23685.724} C_VEL
LIN {X 0,Y 157.451,Z 388.039,A -85,B 0,C 180,E1 -23690.922,E2 -23690.922} C_VEL
LIN {X 0,Y 160.311,Z 384.712,A -85,B 0,C 180,E1 -23696.002,E2 -23696.002} C_VEL
LIN {X 0,Y 164.27,Z 379.869,A -85,B 0,C 180,E1 -23700.891,E2 -23700.891} C_VEL
LIN {X 0,Y 167.94,Z 375.171,A -85,B 0,C 180,E1 -23704.399,E2 -23704.399} C_VEL
LIN {X 0,Y 172.966,Z 368.313,A -85,B 0,C 180,E1 -23708.29,E2 -23708.29} C_VEL
LIN {X 0,Y 178.576,Z 359.766,A -85,B 0,C 180,E1 -23711.994,E2 -23711.994} C_VEL
LIN {X 0,Y 183.975,Z 350.812,A -85,B 0,C 180,E1 -23714.969,E2 -23714.969} C_VEL
LIN {X 0,Y 188.939,Z 341.907,A -85,B 0,C 180,E1 -23717.278,E2 -23717.278} C_VEL
LIN {X 0,Y 194.102,Z 331.252,A -85,B 0,C 180,E1 -23719.497,E2 -23719.497} C_VEL
LIN {X 0,Y 198.431,Z 321.038,A -85,B 0,C 180,E1 -23721.187,E2 -23721.187} C_VEL
LIN {X 0,Y 202.411,Z 310.332,A -85,B 0,C 180,E1 -23722.585,E2 -23722.585} C_VEL
LIN {X 0,Y 206.447,Z 296.854,A -85,B 0,C 180,E1 -23723.951,E2 -23723.951} C_VEL
LIN {X 0,Y 209.573,Z 282.676,A -85,B 0,C 180,E1 -23725.04,E2 -23725.04} C_VEL
LIN {X 0,Y 211.831,Z 268.868,A -85,B 0,C 180,E1 -23725.727,E2 -23725.727} C_VEL
LIN {X 0,Y 213.635,Z 248.341,A -85,B 0,C 180,E1 -23726.38,E2 -23726.38} C_VEL
LIN {X 0,Y 215.961,Z 218.033,A -85,B 0,C 180,E1 -23727.215,E2 -23727.215} C_VEL
LIN {X 0,Y 211.368,Z 207.635,A -85,B 0,C 180,E1 -23729.6,E2 -23729.6} C_VEL
LIN {X 0,Y 205.887,Z 198.058,A -85,B 0,C 180,E1 -23732.627,E2 -23732.627} C_VEL
LIN {X 0,Y 201.043,Z 190.537,A -85,B 0,C 180,E1 -23735.638,E2 -23735.638} C_VEL
LIN {X 0,Y 198.164,Z 186.317,A -85,B 0,C 180,E1 -23737.64,E2 -23737.64} C_VEL
LIN {X 0,Y 195.763,Z 182.843,A -85,B 0,C 180,E1 -23739.476,E2 -23739.476} C_VEL
LIN {X 0,Y 192.753,Z 178.65,A -85,B 0,C 180,E1 -23742.053,E2 -23742.053} C_VEL
LIN {X 0,Y 190.058,Z 174.996,A -85,B 0,C 180,E1 -23744.724,E2 -23744.724} C_VEL
LIN {X 0,Y 189.252,Z 173.868,A -85,B 0,C 180,E1 -23745.62,E2 -23745.62} C_VEL
LIN {X 0,Y 186.833,Z 171.004,A -85,B 0,C 180,E1 -23748.61,E2 -23748.61} C_VEL
LIN {X 0,Y 185.816,Z 168.972,A -85,B 0,C 180,E1 -23750.241,E2 -23750.241} C_VEL
LIN {X 0,Y 182.833,Z 165.897,A -85,B 0,C 180,E1 -23756.453,E2 -23756.453} C_VEL
LIN {X 0,Y 182.3,Z 163.524,A -85,B 0,C 180,E1 -23759.447,E2 -23759.447} C_VEL
LIN {X 0,Y 182.268,Z 163.7,A -85,B 0,C 180,E1 -23766.225,E2 -23766.225} C_VEL
LIN {X 0,Y 183.549,Z 167.282,A -85,B 0,C 180,E1 -23771.386,E2 -23771.386} C_VEL
LIN {X 0,Y 185.93,Z 169.272,A -85,B 0,C 180,E1 -23775.694,E2 -23775.694} C_VEL
LIN {X 0,Y 187.921,Z 172.681,A -85,B 0,C 180,E1 -23778.594,E2 -23778.594} C_VEL
LIN {X 0,Y 189.859,Z 174.677,A -85,B 0,C 180,E1 -23780.783,E2 -23780.783} C_VEL
LIN {X 0,Y 192.584,Z 178.465,A -85,B 0,C 180,E1 -23783.524,E2 -23783.524} C_VEL
LIN {X 0,Y 193.918,Z 180.341,A -85,B 0,C 180,E1 -23784.723,E2 -23784.723} C_VEL
LIN {X 0,Y 196.582,Z 184.054,A -85,B 0,C 180,E1 -23786.901,E2 -23786.901} C_VEL
LIN {X 0,Y 200.687,Z 191.169,A -85,B 0,C 180,E1 -23789.942,E2 -23789.942} C_VEL
LIN {X 0,Y 205.694,Z 200.617,A -85,B 0,C 180,E1 -23793.183,E2 -23793.183} C_VEL
LIN {X 0,Y 210.88,Z 211.535,A -85,B 0,C 180,E1 -23796.164,E2 -23796.164} C_VEL
LIN {X 0,Y 215.614,Z 223.058,A -85,B 0,C 180,E1 -23798.666,E2 -23798.666} C_VEL
LIN {X 0,Y 211.789,Z 272.081,A -85,B 0,C 180,E1 -23800.078,E2 -23800.078} C_VEL
LIN {X 0,Y 209.528,Z 286.51,A -85,B 0,C 180,E1 -23800.725,E2 -23800.725} C_VEL
LIN {X 0,Y 206.367,Z 300.439,A -85,B 0,C 180,E1 -23801.66,E2 -23801.66} C_VEL
LIN {X 0,Y 202.553,Z 313.391,A -85,B 0,C 180,E1 -23802.863,E2 -23802.863} C_VEL
LIN {X 0,Y 197.97,Z 325.96,A -85,B 0,C 180,E1 -23804.402,E2 -23804.402} C_VEL
LIN {X 0,Y 193.046,Z 337.43,A -85,B 0,C 180,E1 -23806.234,E2 -23806.234} C_VEL
LIN {X 0,Y 192.246,Z 339.238,A -85,B 0,C 180,E1 -23806.57,E2 -23806.57} C_VEL
LIN {X 0,Y 189.581,Z 343.845,A -85,B 0,C 180,E1 -23807.343,E2 -23807.343} C_VEL
LIN {X 0,Y 183.7,Z 351.062,A -85,B 0,C 180,E1 -23808.397,E2 -23808.397} C_VEL
LIN {X 0,Y 177.619,Z 357.851,A -85,B 0,C 180,E1 -23809.647,E2 -23809.647} C_VEL
LIN {X 0,Y 174.691,Z 361.717,A -85,B 0,C 180,E1 -23810.733,E2 -23810.733} C_VEL
LIN {X 0,Y 169.296,Z 369.714,A -85,B 0,C 180,E1 -23813.732,E2 -23813.732} C_VEL
LIN {X 0,Y 163.629,Z 377.49,A -85,B 0,C 180,E1 -23817.528,E2 -23817.528} C_VEL
LIN {X 0,Y 159.38,Z 382.944,A -85,B 0,C 180,E1 -23820.984,E2 -23820.984} C_VEL
LIN {X 0,Y 156.077,Z 387.01,A -85,B 0,C 180,E1 -23824.234,E2 -23824.234} C_VEL
LIN {X 0,Y 152.901,Z 390.979,A -85,B 0,C 180,E1 -23828.425,E2 -23828.425} C_VEL
LIN {X 0,Y 149.938,Z 394.465,A -85,B 0,C 180,E1 -23833.666,E2 -23833.666} C_VEL
LIN {X 0,Y 148.277,Z 396.58,A -85,B 0,C 180,E1 -23839.071,E2 -23839.071} C_VEL
LIN {X 0,Y 147.613,Z 397.369,A -85,B 0,C 180,E1 -23844.535,E2 -23844.535} C_VEL
LIN {X 0,Y 147.656,Z 396.833,A -85,B 0,C 180,E1 -23850,E2 -23850} C_VEL
LIN {X 0,Y 147.606,Z 394.926,A -85,B 0,C 180,E1 -23855.464,E2 -23855.464} C_VEL
LIN {X 0,Y 148.205,Z 391.59,A -85,B 0,C 180,E1 -23860.934,E2 -23860.934} C_VEL
LIN {X 0,Y 149.688,Z 386.73,A -85,B 0,C 180,E1 -23866.362,E2 -23866.362} C_VEL
LIN {X 0,Y 151.648,Z 382.048,A -85,B 0,C 180,E1 -23870.339,E2 -23870.339} C_VEL
LIN {X 0,Y 154.561,Z 375.212,A -85,B 0,C 180,E1 -23874.872,E2 -23874.872} C_VEL
LIN {X 0,Y 158.418,Z 366.71,A -85,B 0,C 180,E1 -23879.209,E2 -23879.209} C_VEL
LIN {X 0,Y 162.41,Z 357.839,A -85,B 0,C 180,E1 -23882.745,E2 -23882.745} C_VEL
LIN {X 0,Y 167.091,Z 347.09,A -85,B 0,C 180,E1 -23886.075,E2 -23886.075} C_VEL
LIN {X 0,Y 171.273,Z 336.339,A -85,B 0,C 180,E1 -23888.696,E2 -23888.696} C_VEL
LIN {X 0,Y 175.383,Z 324.289,A -85,B 0,C 180,E1 -23891.009,E2 -23891.009} C_VEL
LIN {X 0,Y 179.323,Z 311.124,A -85,B 0,C 180,E1 -23892.918,E2 -23892.918} C_VEL
LIN {X 0,Y 182.695,Z 297.222,A -85,B 0,C 180,E1 -23894.398,E2 -23894.398} C_VEL
LIN {X 0,Y 185.143,Z 283.317,A -85,B 0,C 180,E1 -23895.473,E2 -23895.473} C_VEL
LIN {X 0,Y 186.961,Z 268.399,A -85,B 0,C 180,E1 -23896.195,E2 -23896.195} C_VEL
LIN {X 0,Y 190.93,Z 207.974,A -85,B 0,C 180,E1 -23898.199,E2 -23898.199} C_VEL
LIN {X 0,Y 186.015,Z 194.831,A -85,B 0,C 180,E1 -23900.477,E2 -23900.477} C_VEL
LIN {X 0,Y 180.462,Z 182.505,A -85,B 0,C 180,E1 -23903.182,E2 -23903.182} C_VEL
LIN {X 0,Y 176.06,Z 174.042,A -85,B 0,C 180,E1 -23905.483,E2 -23905.483} C_VEL
LIN {X 0,Y 170.119,Z 165.279,A -85,B 0,C 180,E1 -23908.811,E2 -23908.811} C_VEL
LIN {X 0,Y 166.331,Z 160.295,A -85,B 0,C 180,E1 -23911.177,E2 -23911.177} C_VEL
LIN {X 0,Y 163.256,Z 156.161,A -85,B 0,C 180,E1 -23913.313,E2 -23913.313} C_VEL
LIN {X 0,Y 160.634,Z 153.198,A -85,B 0,C 180,E1 -23915.268,E2 -23915.268} C_VEL
LIN {X 0,Y 159.447,Z 151.187,A -85,B 0,C 180,E1 -23916.284,E2 -23916.284} C_VEL
LIN {X 0,Y 156.841,Z 148.936,A -85,B 0,C 180,E1 -23918.477,E2 -23918.477} C_VEL
LIN {X 0,Y 155.319,Z 146.051,A -85,B 0,C 180,E1 -23920.066,E2 -23920.066} C_VEL
LIN {X 0,Y 154.886,Z 145.636,A -85,B 0,C 180,E1 -23920.495,E2 -23920.495} C_VEL
LIN {X 0,Y 152.139,Z 143.706,A -85,B 0,C 180,E1 -23923.392,E2 -23923.392} C_VEL
LIN {X 0,Y 150.786,Z 141.349,A -85,B 0,C 180,E1 -23925.233,E2 -23925.233} C_VEL
LIN {X 0,Y 150.433,Z 139.856,A -85,B 0,C 180,E1 -23925.975,E2 -23925.975} C_VEL
LIN {X 0,Y 150.648,Z 139.83,A -85,B 0,C 180,E1 -23929.246,E2 -23929.246} C_VEL
LIN {X 0,Y 150.74,Z 139.825,A -85,B 0,C 180,E1 -23931.96,E2 -23931.96} C_VEL
LIN {X 0,Y 151.217,Z 139.752,A -85,B 0,C 180,E1 -23940,E2 -23940} C_VEL
LIN {X 0,Y 150.685,Z 139.82,A -85,B 0,C 180,E1 -23948.044,E2 -23948.044} C_VEL
LIN {X 0,Y 150.576,Z 139.827,A -85,B 0,C 180,E1 -23951.437,E2 -23951.437} C_VEL
LIN {X 0,Y 150.374,Z 139.855,A -85,B 0,C 180,E1 -23956.286,E2 -23956.286} C_VEL
LIN {X 0,Y 150.427,Z 140.019,A -85,B 0,C 180,E1 -23960.503,E2 -23960.503} C_VEL
LIN {X 0,Y 151.07,Z 142.257,A -85,B 0,C 180,E1 -23961.606,E2 -23961.606} C_VEL
LIN {X 0,Y 152.775,Z 144.447,A -85,B 0,C 180,E1 -23963.736,E2 -23963.736} C_VEL
LIN {X 0,Y 155.258,Z 145.985,A -85,B 0,C 180,E1 -23966.246,E2 -23966.246} C_VEL
LIN {X 0,Y 156.826,Z 148.974,A -85,B 0,C 180,E1 -23967.889,E2 -23967.889} C_VEL
LIN {X 0,Y 159.184,Z 151.05,A -85,B 0,C 180,E1 -23969.889,E2 -23969.889} C_VEL
LIN {X 0,Y 159.858,Z 151.861,A -85,B 0,C 180,E1 -23970.445,E2 -23970.445} C_VEL
LIN {X 0,Y 162.118,Z 155.145,A -85,B 0,C 180,E1 -23972.261,E2 -23972.261} C_VEL
LIN {X 0,Y 163.831,Z 156.964,A -85,B 0,C 180,E1 -23973.482,E2 -23973.482} C_VEL
LIN {X 0,Y 166.67,Z 160.712,A -85,B 0,C 180,E1 -23975.419,E2 -23975.419} C_VEL
LIN {X 0,Y 171.391,Z 167.347,A -85,B 0,C 180,E1 -23978.333,E2 -23978.333} C_VEL
LIN {X 0,Y 175.964,Z 174.065,A -85,B 0,C 180,E1 -23980.852,E2 -23980.852} C_VEL
LIN {X 0,Y 181.895,Z 183.571,A -85,B 0,C 180,E1 -23983.796,E2 -23983.796} C_VEL
LIN {X 0,Y 188.458,Z 195.913,A -85,B 0,C 180,E1 -23986.761,E2 -23986.761} C_VEL
LIN {X 0,Y 191.229,Z 202.704,A -85,B 0,C 180,E1 -23987.991,E2 -23987.991} C_VEL
LIN {X 0,Y 186.97,Z 265.631,A -85,B 0,C 180,E1 -23990.078,E2 -23990.078} C_VEL
LIN {X 0,Y 185.247,Z 279.741,A -85,B 0,C 180,E1 -23990.897,E2 -23990.897} C_VEL
LIN {X 0,Y 182.78,Z 293.25,A -85,B 0,C 180,E1 -23992.034,E2 -23992.034} C_VEL
LIN {X 0,Y 179.895,Z 305.535,A -85,B 0,C 180,E1 -23993.433,E2 -23993.433} C_VEL
LIN {X 0,Y 176.086,Z 318.412,A -85,B 0,C 180,E1 -23995.338,E2 -23995.338} C_VEL
LIN {X 0,Y 172.216,Z 330.07,A -85,B 0,C 180,E1 -23997.615,E2 -23997.615} C_VEL
LIN {X 0,Y 168.52,Z 339.785,A -85,B 0,C 180,E1 -23999.971,E2 -23999.971} C_VEL
LIN {X 0,Y 163.942,Z 350.53,A -85,B 0,C 180,E1 -24003.249,E2 -24003.249} C_VEL
LIN {X 0,Y 159.924,Z 359.401,A -85,B 0,C 180,E1 -24006.702,E2 -24006.702} C_VEL
LIN {X 0,Y 156.059,Z 367.89,A -85,B 0,C 180,E1 -24010.944,E2 -24010.944} C_VEL
LIN {X 0,Y 152.645,Z 375.223,A -85,B 0,C 180,E1 -24015.694,E2 -24015.694} C_VEL
LIN {X 0,Y 150.181,Z 380.897,A -85,B 0,C 180,E1 -24020.574,E2 -24020.574} C_VEL
LIN {X 0,Y 148.825,Z 384.406,A -85,B 0,C 180,E1 -24024.581,E2 -24024.581} C_VEL
LIN {X 0,Y 147.836,Z 387.846,A -85,B 0,C 180,E1 -24030,E2 -24030} C_VEL
LIN {X 0,Y 147.642,Z 389.046,A -85,B 0,C 180,E1 -24032.729,E2 -24032.729} C_VEL
LIN {X 0,Y 147.523,Z 389.914,A -85,B 0,C 180,E1 -24035.468,E2 -24035.468} C_VEL
LIN {X 0,Y 147.633,Z 390.663,A -85,B 0,C 180,E1 -24040.978,E2 -24040.978} C_VEL
LIN {X 0,Y 148.698,Z 390.074,A -85,B 0,C 180,E1 -24046.474,E2 -24046.474} C_VEL
LIN {X 0,Y 150.708,Z 388.121,A -85,B 0,C 180,E1 -24051.905,E2 -24051.905} C_VEL
LIN {X 0,Y 153.826,Z 384.754,A -85,B 0,C 180,E1 -24057.186,E2 -24057.186} C_VEL
LIN {X 0,Y 158.087,Z 379.869,A -85,B 0,C 180,E1 -24062.241,E2 -24062.241} C_VEL
LIN {X 0,Y 162.014,Z 375.125,A -85,B 0,C 180,E1 -24065.847,E2 -24065.847} C_VEL
LIN {X 0,Y 167.34,Z 368.218,A -85,B 0,C 180,E1 -24069.828,E2 -24069.828} C_VEL
LIN {X 0,Y 173.256,Z 359.615,A -85,B 0,C 180,E1 -24073.598,E2 -24073.598} C_VEL
LIN {X 0,Y 178.95,Z 350.6,A -85,B 0,C 180,E1 -24076.599,E2 -24076.599} C_VEL
LIN {X 0,Y 185.203,Z 339.655,A -85,B 0,C 180,E1 -24079.372,E2 -24079.372} C_VEL
LIN {X 0,Y 190.565,Z 328.502,A -85,B 0,C 180,E1 -24081.6,E2 -24081.6} C_VEL
LIN {X 0,Y 195.238,Z 317.677,A -85,B 0,C 180,E1 -24083.22,E2 -24083.22} C_VEL
LIN {X 0,Y 199.893,Z 304.301,A -85,B 0,C 180,E1 -24084.83,E2 -24084.83} C_VEL
LIN {X 0,Y 203.464,Z 291.305,A -85,B 0,C 180,E1 -24085.997,E2 -24085.997} C_VEL
LIN {X 0,Y 206.315,Z 277.184,A -85,B 0,C 180,E1 -24086.922,E2 -24086.922} C_VEL
LIN {X 0,Y 208.306,Z 262.791,A -85,B 0,C 180,E1 -24087.509,E2 -24087.509} C_VEL
LIN {X 0,Y 211.674,Z 220.904,A -85,B 0,C 180,E1 -24088.684,E2 -24088.684} C_VEL
LIN {X 0,Y 207.8,Z 212.002,A -85,B 0,C 180,E1 -24090.841,E2 -24090.841} C_VEL
LIN {X 0,Y 202.914,Z 203.344,A -85,B 0,C 180,E1 -24093.713,E2 -24093.713} C_VEL
LIN {X 0,Y 198.492,Z 196.228,A -85,B 0,C 180,E1 -24096.637,E2 -24096.637} C_VEL
LIN {X 0,Y 194.122,Z 189.542,A -85,B 0,C 180,E1 -24099.986,E2 -24099.986} C_VEL
LIN {X 0,Y 190.894,Z 185.022,A -85,B 0,C 180,E1 -24102.87,E2 -24102.87} C_VEL
LIN {X 0,Y 188.23,Z 181.06,A -85,B 0,C 180,E1 -24105.713,E2 -24105.713} C_VEL
LIN {X 0,Y 185.489,Z 177.689,A -85,B 0,C 180,E1 -24109.223,E2 -24109.223} C_VEL
LIN {X 0,Y 184.506,Z 175.79,A -85,B 0,C 180,E1 -24110.881,E2 -24110.881} C_VEL
LIN {X 0,Y 181.744,Z 172.587,A -85,B 0,C 180,E1 -24117.229,E2 -24117.229} C_VEL
LIN {X 0,Y 181.345,Z 170.488,A -85,B 0,C 180,E1 -24120,E2 -24120} C_VEL
LIN {X 0,Y 181.347,Z 170.687,A -85,B 0,C 180,E1 -24125.888,E2 -24125.888} C_VEL
LIN {X 0,Y 182.548,Z 174.25,A -85,B 0,C 180,E1 -24131.098,E2 -24131.098} C_VEL
LIN {X 0,Y 184.734,Z 176.233,A -85,B 0,C 180,E1 -24135.254,E2 -24135.254} C_VEL
LIN {X 0,Y 186.691,Z 179.543,A -85,B 0,C 180,E1 -24138.208,E2 -24138.208} C_VEL
LIN {X 0,Y 188.406,Z 181.472,A -85,B 0,C 180,E1 -24140.238,E2 -24140.238} C_VEL
LIN {X 0,Y 191.26,Z 185.396,A -85,B 0,C 180,E1 -24143.196,E2 -24143.196} C_VEL
LIN {X 0,Y 194.547,Z 190.329,A -85,B 0,C 180,E1 -24146.108,E2 -24146.108} C_VEL
LIN {X 0,Y 198.763,Z 197.895,A -85,B 0,C 180,E1 -24149.38,E2 -24149.38} C_VEL
LIN {X 0,Y 203.629,Z 207.651,A -85,B 0,C 180,E1 -24152.672,E2 -24152.672} C_VEL
LIN {X 0,Y 208.336,Z 218.219,A -85,B 0,C 180,E1 -24155.511,E2 -24155.511} C_VEL
LIN {X 0,Y 211.259,Z 225.553,A -85,B 0,C 180,E1 -24157.154,E2 -24157.154} C_VEL
LIN {X 0,Y 207.607,Z 271.641,A -85,B 0,C 180,E1 -24158.507,E2 -24158.507} C_VEL
LIN {X 0,Y 205.296,Z 286.045,A -85,B 0,C 180,E1 -24159.14,E2 -24159.14} C_VEL
LIN {X 0,Y 202.054,Z 300.05,A -85,B 0,C 180,E1 -24160.073,E2 -24160.073} C_VEL
LIN {X 0,Y 197.822,Z 313.929,A -85,B 0,C 180,E1 -24161.365,E2 -24161.365} C_VEL
LIN {X 0,Y 193.084,Z 326.363,A -85,B 0,C 180,E1 -24162.901,E2 -24162.901} C_VEL
LIN {X 0,Y 187.452,Z 338.901,A -85,B 0,C 180,E1 -24164.954,E2 -24164.954} C_VEL
LIN {X 0,Y 181.407,Z 350.511,A -85,B 0,C 180,E1 -24167.491,E2 -24167.491} C_VEL
LIN {X 0,Y 175.723,Z 360.13,A -85,B 0,C 180,E1 -24170.214,E2 -24170.214} C_VEL
LIN {X 0,Y 174.691,Z 361.717,A -85,B 0,C 180,E1 -24170.733,E2 -24170.733} C_VEL
LIN {X 0,Y 171.739,Z 365.461,A -85,B 0,C 180,E1 -24171.901,E2 -24171.901} C_VEL
LIN {X 0,Y 165.432,Z 371.205,A -85,B 0,C 180,E1 -24173.64,E2 -24173.64} C_VEL
LIN {X 0,Y 159.14,Z 376.395,A -85,B 0,C 180,E1 -24175.628,E2 -24175.628} C_VEL
LIN {X 0,Y 156.278,Z 379.246,A -85,B 0,C 180,E1 -24177.175,E2 -24177.175} C_VEL
LIN {X 0,Y 151.809,Z 384.554,A -85,B 0,C 180,E1 -24180.915,E2 -24180.915} C_VEL
LIN {X 0,Y 148.285,Z 388.651,A -85,B 0,C 180,E1 -24184.75,E2 -24184.75} C_VEL
LIN {X 0,Y 144.564,Z 392.823,A -85,B 0,C 180,E1 -24190.104,E2 -24190.104} C_VEL
LIN {X 0,Y 142.039,Z 395.581,A -85,B 0,C 180,E1 -24195.676,E2 -24195.676} C_VEL
LIN {X 0,Y 140.771,Z 396.999,A -85,B 0,C 180,E1 -24201.386,E2 -24201.386} C_VEL
LIN {X 0,Y 140.485,Z 397.096,A -85,B 0,C 180,E1 -24207.132,E2 -24207.132} C_VEL
LIN {X 0,Y 140.559,Z 396.643,A -85,B 0,C 180,E1 -24210,E2 -24210} C_VEL
LIN {X 0,Y 140.484,Z 395.844,A -85,B 0,C 180,E1 -24212.867,E2 -24212.867} C_VEL
LIN {X 0,Y 140.745,Z 393.19,A -85,B 0,C 180,E1 -24218.615,E2 -24218.615} C_VEL
LIN {X 0,Y 141.857,Z 389.069,A -85,B 0,C 180,E1 -24224.342,E2 -24224.342} C_VEL
LIN {X 0,Y 144.211,Z 383.372,A -85,B 0,C 180,E1 -24229.946,E2 -24229.946} C_VEL
LIN {X 0,Y 147.139,Z 376.748,A -85,B 0,C 180,E1 -24234.836,E2 -24234.836} C_VEL
LIN {X 0,Y 150.962,Z 368.914,A -85,B 0,C 180,E1 -24239.263,E2 -24239.263} C_VEL
LIN {X 0,Y 154.927,Z 360.52,A -85,B 0,C 180,E1 -24242.98,E2 -24242.98} C_VEL
LIN {X 0,Y 159.702,Z 350.421,A -85,B 0,C 180,E1 -24246.447,E2 -24246.447} C_VEL
LIN {X 0,Y 164.026,Z 340.243,A -85,B 0,C 180,E1 -24249.196,E2 -24249.196} C_VEL
LIN {X 0,Y 168.575,Z 327.871,A -85,B 0,C 180,E1 -24251.839,E2 -24251.839} C_VEL
LIN {X 0,Y 172.572,Z 315.596,A -85,B 0,C 180,E1 -24253.814,E2 -24253.814} C_VEL
LIN {X 0,Y 176.279,Z 301.948,A -85,B 0,C 180,E1 -24255.45,E2 -24255.45} C_VEL
LIN {X 0,Y 179.264,Z 287.601,A -85,B 0,C 180,E1 -24256.697,E2 -24256.697} C_VEL
LIN {X 0,Y 181.306,Z 273.508,A -85,B 0,C 180,E1 -24257.524,E2 -24257.524} C_VEL
LIN {X 0,Y 183.16,Z 250.196,A -85,B 0,C 180,E1 -24258.343,E2 -24258.343} C_VEL
LIN {X 0,Y 185.823,Z 209.935,A -85,B 0,C 180,E1 -24259.7,E2 -24259.7} C_VEL
LIN {X 0,Y 181.681,Z 198.68,A -85,B 0,C 180,E1 -24261.762,E2 -24261.762} C_VEL
LIN {X 0,Y 176.327,Z 186.501,A -85,B 0,C 180,E1 -24264.563,E2 -24264.563} C_VEL
LIN {X 0,Y 172.416,Z 178.852,A -85,B 0,C 180,E1 -24266.756,E2 -24266.756} C_VEL
LIN {X 0,Y 167.074,Z 170.856,A -85,B 0,C 180,E1 -24269.945,E2 -24269.945} C_VEL
LIN {X 0,Y 163.624,Z 166.158,A -85,B 0,C 180,E1 -24272.238,E2 -24272.238} C_VEL
LIN {X 0,Y 160.865,Z 162.362,A -85,B 0,C 180,E1 -24274.269,E2 -24274.269} C_VEL
LIN {X 0,Y 158.22,Z 159.113,A -85,B 0,C 180,E1 -24276.382,E2 -24276.382} C_VEL
LIN {X 0,Y 157.347,Z 157.676,A -85,B 0,C 180,E1 -24277.168,E2 -24277.168} C_VEL
LIN {X 0,Y 154.656,Z 154.983,A -85,B 0,C 180,E1 -24279.608,E2 -24279.608} C_VEL
LIN {X 0,Y 153.15,Z 152.366,A -85,B 0,C 180,E1 -24281.263,E2 -24281.263} C_VEL
LIN {X 0,Y 150.489,Z 150.274,A -85,B 0,C 180,E1 -24284.25,E2 -24284.25} C_VEL
LIN {X 0,Y 148.915,Z 147.198,A -85,B 0,C 180,E1 -24286.612,E2 -24286.612} C_VEL
LIN {X 0,Y 148.665,Z 146.709,A -85,B 0,C 180,E1 -24287.024,E2 -24287.024} C_VEL
LIN {X 0,Y 145.076,Z 144.21,A -85,B 0,C 180,E1 -24293.743,E2 -24293.743} C_VEL
LIN {X 0,Y 144.133,Z 141.966,A -85,B 0,C 180,E1 -24297.38,E2 -24297.38} C_VEL
LIN {X 0,Y 144.014,Z 140.662,A -85,B 0,C 180,E1 -24298.952,E2 -24298.952} C_VEL
LIN {X 0,Y 144.175,Z 140.628,A -85,B 0,C 180,E1 -24300,E2 -24300} C_VEL
LIN {X 0,Y 143.654,Z 140.924,A -85,B 0,C 180,E1 -24305.616,E2 -24305.616} C_VEL
LIN {X 0,Y 146.381,Z 145.713,A -85,B 0,C 180,E1 -24315.669,E2 -24315.669} C_VEL
LIN {X 0,Y 148.798,Z 147.009,A -85,B 0,C 180,E1 -24319.574,E2 -24319.574} C_VEL
LIN {X 0,Y 150.059,Z 149.816,A -85,B 0,C 180,E1 -24321.569,E2 -24321.569} C_VEL
LIN {X 0,Y 152.539,Z 152.112,A -85,B 0,C 180,E1 -24324.498,E2 -24324.498} C_VEL
LIN {X 0,Y 153.453,Z 152.792,A -85,B 0,C 180,E1 -24325.443,E2 -24325.443} C_VEL
LIN {X 0,Y 155.184,Z 155.727,A -85,B 0,C 180,E1 -24327.294,E2 -24327.294} C_VEL
LIN {X 0,Y 157.672,Z 158.2,A -85,B 0,C 180,E1 -24329.502,E2 -24329.502} C_VEL
LIN {X 0,Y 160.123,Z 161.662,A -85,B 0,C 180,E1 -24331.555,E2 -24331.555} C_VEL
LIN {X 0,Y 161.619,Z 163.48,A -85,B 0,C 180,E1 -24332.689,E2 -24332.689} C_VEL
LIN {X 0,Y 165.322,Z 168.573,A -85,B 0,C 180,E1 -24335.305,E2 -24335.305} C_VEL
LIN {X 0,Y 168.627,Z 173.32,A -85,B 0,C 180,E1 -24337.416,E2 -24337.416} C_VEL
LIN {X 0,Y 172.937,Z 179.893,A -85,B 0,C 180,E1 -24339.925,E2 -24339.925} C_VEL
LIN {X 0,Y 178.469,Z 189.07,A -85,B 0,C 180,E1 -24342.83,E2 -24342.83} C_VEL
LIN {X 0,Y 184.407,Z 200.537,A -85,B 0,C 180,E1 -24345.676,E2 -24345.676} C_VEL
LIN {X 0,Y 186.149,Z 204.821,A -85,B 0,C 180,E1 -24346.5,E2 -24346.5} C_VEL
LIN {X 0,Y 181.849,Z 265.962,A -85,B 0,C 180,E1 -24348.559,E2 -24348.559} C_VEL
LIN {X 0,Y 179.967,Z 280.524,A -85,B 0,C 180,E1 -24349.425,E2 -24349.425} C_VEL
LIN {X 0,Y 177.285,Z 294.434,A -85,B 0,C 180,E1 -24350.634,E2 -24350.634} C_VEL
LIN {X 0,Y 174.269,Z 306.5,A -85,B 0,C 180,E1 -24352.048,E2 -24352.048} C_VEL
LIN {X 0,Y 170.335,Z 319.221,A -85,B 0,C 180,E1 -24353.989,E2 -24353.989} C_VEL
LIN {X 0,Y 166.303,Z 330.767,A -85,B 0,C 180,E1 -24356.313,E2 -24356.313} C_VEL
LIN {X 0,Y 162.436,Z 340.393,A -85,B 0,C 180,E1 -24358.722,E2 -24358.722} C_VEL
LIN {X 0,Y 157.676,Z 351.062,A -85,B 0,C 180,E1 -24362.095,E2 -24362.095} C_VEL
LIN {X 0,Y 153.444,Z 359.873,A -85,B 0,C 180,E1 -24365.656,E2 -24365.656} C_VEL
LIN {X 0,Y 149.398,Z 368.307,A -85,B 0,C 180,E1 -24370.059,E2 -24370.059} C_VEL
LIN {X 0,Y 146.023,Z 375.085,A -85,B 0,C 180,E1 -24374.628,E2 -24374.628} C_VEL
LIN {X 0,Y 143.692,Z 379.818,A -85,B 0,C 180,E1 -24378.718,E2 -24378.718} C_VEL
LIN {X 0,Y 142.229,Z 383.628,A -85,B 0,C 180,E1 -24382.904,E2 -24382.904} C_VEL
LIN {X 0,Y 141.133,Z 386.568,A -85,B 0,C 180,E1 -24387.146,E2 -24387.146} C_VEL
LIN {X 0,Y 140.542,Z 389.273,A -85,B 0,C 180,E1 -24392.867,E2 -24392.867} C_VEL
LIN {X 0,Y 140.416,Z 390.124,A -85,B 0,C 180,E1 -24395.746,E2 -24395.746} C_VEL
LIN {X 0,Y 140.592,Z 390.832,A -85,B 0,C 180,E1 -24401.535,E2 -24401.535} C_VEL
LIN {X 0,Y 141.792,Z 390.197,A -85,B 0,C 180,E1 -24407.301,E2 -24407.301} C_VEL
LIN {X 0,Y 144.036,Z 388.202,A -85,B 0,C 180,E1 -24412.977,E2 -24412.977} C_VEL
LIN {X 0,Y 147.416,Z 384.795,A -85,B 0,C 180,E1 -24418.473,E2 -24418.473} C_VEL
LIN {X 0,Y 152.006,Z 379.869,A -85,B 0,C 180,E1 -24423.699,E2 -24423.699} C_VEL
LIN {X 0,Y 156.202,Z 375.081,A -85,B 0,C 180,E1 -24427.403,E2 -24427.403} C_VEL
LIN {X 0,Y 161.849,Z 368.126,A -85,B 0,C 180,E1 -24431.469,E2 -24431.469} C_VEL
LIN {X 0,Y 168.088,Z 359.469,A -85,B 0,C 180,E1 -24435.3,E2 -24435.3} C_VEL
LIN {X 0,Y 174.088,Z 350.392,A -85,B 0,C 180,E1 -24438.319,E2 -24438.319} C_VEL
LIN {X 0,Y 180.607,Z 339.373,A -85,B 0,C 180,E1 -24441.102,E2 -24441.102} C_VEL
LIN {X 0,Y 186.19,Z 328.113,A -85,B 0,C 180,E1 -24443.332,E2 -24443.332} C_VEL
LIN {X 0,Y 191.641,Z 315.634,A -85,B 0,C 180,E1 -24445.141,E2 -24445.141} C_VEL
LIN {X 0,Y 195.859,Z 303.561,A -85,B 0,C 180,E1 -24446.541,E2 -24446.541} C_VEL
LIN {X 0,Y 199.529,Z 290.276,A -85,B 0,C 180,E1 -24447.71,E2 -24447.71} C_VEL
LIN {X 0,Y 202.28,Z 276.943,A -85,B 0,C 180,E1 -24448.557,E2 -24448.557} C_VEL
LIN {X 0,Y 204.299,Z 262.435,A -85,B 0,C 180,E1 -24449.141,E2 -24449.141} C_VEL
LIN {X 0,Y 207.509,Z 223.764,A -85,B 0,C 180,E1 -24450.224,E2 -24450.224} C_VEL
LIN {X 0,Y 204.344,Z 216.486,A -85,B 0,C 180,E1 -24452.112,E2 -24452.112} C_VEL
LIN {X 0,Y 199.822,Z 208.238,A -85,B 0,C 180,E1 -24454.964,E2 -24454.964} C_VEL
LIN {X 0,Y 195.835,Z 201.603,A -85,B 0,C 180,E1 -24457.793,E2 -24457.793} C_VEL
LIN {X 0,Y 191.736,Z 195.292,A -85,B 0,C 180,E1 -24461.154,E2 -24461.154} C_VEL
LIN {X 0,Y 189.105,Z 191.396,A -85,B 0,C 180,E1 -24463.676,E2 -24463.676} C_VEL
LIN {X 0,Y 186.486,Z 187.42,A -85,B 0,C 180,E1 -24466.654,E2 -24466.654} C_VEL
LIN {X 0,Y 184.079,Z 184.193,A -85,B 0,C 180,E1 -24469.994,E2 -24469.994} C_VEL
LIN {X 0,Y 183.429,Z 182.737,A -85,B 0,C 180,E1 -24471.184,E2 -24471.184} C_VEL
LIN {X 0,Y 180.798,Z 179.585,A -85,B 0,C 180,E1 -24477.493,E2 -24477.493} C_VEL
LIN {X 0,Y 180.455,Z 177.718,A -85,B 0,C 180,E1 -24480,E2 -24480} C_VEL
LIN {X 0,Y 180.31,Z 177.631,A -85,B 0,C 180,E1 -24484.471,E2 -24484.471} C_VEL
LIN {X 0,Y 180.46,Z 178.098,A -85,B 0,C 180,E1 -24486.032,E2 -24486.032} C_VEL
LIN {X 0,Y 181.827,Z 181.561,A -85,B 0,C 180,E1 -24491.495,E2 -24491.495} C_VEL
LIN {X 0,Y 183.535,Z 183.164,A -85,B 0,C 180,E1 -24494.783,E2 -24494.783} C_VEL
LIN {X 0,Y 185.471,Z 186.399,A -85,B 0,C 180,E1 -24497.817,E2 -24497.817} C_VEL
LIN {X 0,Y 186.979,Z 188.237,A -85,B 0,C 180,E1 -24499.689,E2 -24499.689} C_VEL
LIN {X 0,Y 190.136,Z 192.887,A -85,B 0,C 180,E1 -24503.081,E2 -24503.081} C_VEL
LIN {X 0,Y 192.551,Z 196.583,A -85,B 0,C 180,E1 -24505.296,E2 -24505.296} C_VEL
LIN {X 0,Y 196.524,Z 204.115,A -85,B 0,C 180,E1 -24508.566,E2 -24508.566} C_VEL
LIN {X 0,Y 201.104,Z 213.731,A -85,B 0,C 180,E1 -24511.84,E2 -24511.84} C_VEL
LIN {X 0,Y 205.442,Z 224.034,A -85,B 0,C 180,E1 -24514.617,E2 -24514.617} C_VEL
LIN {X 0,Y 207.141,Z 228.479,A -85,B 0,C 180,E1 -24515.642,E2 -24515.642} C_VEL
LIN {X 0,Y 203.518,Z 271.646,A -85,B 0,C 180,E1 -24516.886,E2 -24516.886} C_VEL
LIN {X 0,Y 201.072,Z 286.338,A -85,B 0,C 180,E1 -24517.534,E2 -24517.534} C_VEL
LIN {X 0,Y 197.901,Z 299.661,A -85,B 0,C 180,E1 -24518.417,E2 -24518.417} C_VEL
LIN {X 0,Y 193.826,Z 312.713,A -85,B 0,C 180,E1 -24519.6,E2 -24519.6} C_VEL
LIN {X 0,Y 188.977,Z 325.345,A -85,B 0,C 180,E1 -24521.141,E2 -24521.141} C_VEL
LIN {X 0,Y 183.662,Z 336.867,A -85,B 0,C 180,E1 -24522.959,E2 -24522.959} C_VEL
LIN {X 0,Y 177.784,Z 348.033,A -85,B 0,C 180,E1 -24525.283,E2 -24525.283} C_VEL
LIN {X 0,Y 172.346,Z 357.132,A -85,B 0,C 180,E1 -24527.713,E2 -24527.713} C_VEL
LIN {X 0,Y 166.4,Z 365.954,A -85,B 0,C 180,E1 -24530.688,E2 -24530.688} C_VEL
LIN {X 0,Y 160.987,Z 373.308,A -85,B 0,C 180,E1 -24533.888,E2 -24533.888} C_VEL
LIN {X 0,Y 156.278,Z 379.246,A -85,B 0,C 180,E1 -24537.175,E2 -24537.175} C_VEL
LIN {X 0,Y 154.171,Z 381.111,A -85,B 0,C 180,E1 -24538.225,E2 -24538.225} C_VEL
LIN {X 0,Y 144.484,Z 386.335,A -85,B 0,C 180,E1 -24541.251,E2 -24541.251} C_VEL
LIN {X 0,Y 142.616,Z 387.719,A -85,B 0,C 180,E1 -24542.538,E2 -24542.538} C_VEL
LIN {X 0,Y 139.715,Z 390.863,A -85,B 0,C 180,E1 -24546.27,E2 -24546.27} C_VEL
LIN {X 0,Y 136.289,Z 394.28,A -85,B 0,C 180,E1 -24551.976,E2 -24551.976} C_VEL
LIN {X 0,Y 134.279,Z 396.331,A -85,B 0,C 180,E1 -24557.915,E2 -24557.915} C_VEL
LIN {X 0,Y 133.45,Z 397.055,A -85,B 0,C 180,E1 -24563.953,E2 -24563.953} C_VEL
LIN {X 0,Y 133.395,Z 396.92,A -85,B 0,C 180,E1 -24566.979,E2 -24566.979} C_VEL
LIN {X 0,Y 133.473,Z 396.449,A -85,B 0,C 180,E1 -24570,E2 -24570} C_VEL
LIN {X 0,Y 133.395,Z 395.63,A -85,B 0,C 180,E1 -24573.02,E2 -24573.02} C_VEL
LIN {X 0,Y 133.698,Z 392.939,A -85,B 0,C 180,E1 -24579.073,E2 -24579.073} C_VEL
LIN {X 0,Y 134.926,Z 388.782,A -85,B 0,C 180,E1 -24585.096,E2 -24585.096} C_VEL
LIN {X 0,Y 137.484,Z 383.047,A -85,B 0,C 180,E1 -24590.967,E2 -24590.967} C_VEL
LIN {X 0,Y 140.392,Z 376.915,A -85,B 0,C 180,E1 -24595.701,E2 -24595.701} C_VEL
LIN {X 0,Y 144.098,Z 369.749,A -85,B 0,C 180,E1 -24599.994,E2 -24599.994} C_VEL
LIN {X 0,Y 148.222,Z 361.56,A -85,B 0,C 180,E1 -24603.857,E2 -24603.857} C_VEL
LIN {X 0,Y 153.132,Z 351.697,A -85,B 0,C 180,E1 -24607.452,E2 -24607.452} C_VEL
LIN {X 0,Y 157.612,Z 341.807,A -85,B 0,C 180,E1 -24610.282,E2 -24610.282} C_VEL
LIN {X 0,Y 162.237,Z 330.1,A -85,B 0,C 180,E1 -24612.936,E2 -24612.936} C_VEL
LIN {X 0,Y 166.429,Z 318.086,A -85,B 0,C 180,E1 -24615.017,E2 -24615.017} C_VEL
LIN {X 0,Y 170.52,Z 304.257,A -85,B 0,C 180,E1 -24616.801,E2 -24616.801} C_VEL
LIN {X 0,Y 173.735,Z 290.046,A -85,B 0,C 180,E1 -24618.122,E2 -24618.122} C_VEL
LIN {X 0,Y 176.02,Z 275.97,A -85,B 0,C 180,E1 -24619.014,E2 -24619.014} C_VEL
LIN {X 0,Y 177.684,Z 258.173,A -85,B 0,C 180,E1 -24619.696,E2 -24619.696} C_VEL
LIN {X 0,Y 180.864,Z 212.099,A -85,B 0,C 180,E1 -24621.267,E2 -24621.267} C_VEL
LIN {X 0,Y 177.466,Z 202.631,A -85,B 0,C 180,E1 -24623.095,E2 -24623.095} C_VEL
LIN {X 0,Y 172.668,Z 191.328,A -85,B 0,C 180,E1 -24625.792,E2 -24625.792} C_VEL
LIN {X 0,Y 169.031,Z 183.923,A -85,B 0,C 180,E1 -24627.981,E2 -24627.981} C_VEL
LIN {X 0,Y 164.129,Z 176.472,A -85,B 0,C 180,E1 -24631.098,E2 -24631.098} C_VEL
LIN {X 0,Y 160.846,Z 171.827,A -85,B 0,C 180,E1 -24633.432,E2 -24633.432} C_VEL
LIN {X 0,Y 158.486,Z 168.51,A -85,B 0,C 180,E1 -24635.282,E2 -24635.282} C_VEL
LIN {X 0,Y 155.701,Z 164.72,A -85,B 0,C 180,E1 -24637.691,E2 -24637.691} C_VEL
LIN {X 0,Y 152.206,Z 160.469,A -85,B 0,C 180,E1 -24641.143,E2 -24641.143} C_VEL
LIN {X 0,Y 151.409,Z 159.023,A -85,B 0,C 180,E1 -24642.091,E2 -24642.091} C_VEL
LIN {X 0,Y 148.792,Z 156.672,A -85,B 0,C 180,E1 -24645.249,E2 -24645.249} C_VEL
LIN {X 0,Y 147.137,Z 153.492,A -85,B 0,C 180,E1 -24647.938,E2 -24647.938} C_VEL
LIN {X 0,Y 143.962,Z 151.045,A -85,B 0,C 180,E1 -24654.397,E2 -24654.397} C_VEL
LIN {X 0,Y 143.105,Z 148.654,A -85,B 0,C 180,E1 -24658.242,E2 -24658.242} C_VEL
LIN {X 0,Y 143.013,Z 147.762,A -85,B 0,C 180,E1 -24659.297,E2 -24659.297} C_VEL
LIN {X 0,Y 142.745,Z 147.82,A -85,B 0,C 180,E1 -24664.943,E2 -24664.943} C_VEL
LIN {X 0,Y 143.729,Z 150.858,A -85,B 0,C 180,E1 -24671.28,E2 -24671.28} C_VEL
LIN {X 0,Y 145.902,Z 153.072,A -85,B 0,C 180,E1 -24676.443,E2 -24676.443} C_VEL
LIN {X 0,Y 147.29,Z 153.765,A -85,B 0,C 180,E1 -24678.699,E2 -24678.699} C_VEL
LIN {X 0,Y 148.811,Z 156.843,A -85,B 0,C 180,E1 -24681.173,E2 -24681.173} C_VEL
LIN {X 0,Y 151.708,Z 159.537,A -85,B 0,C 180,E1 -24684.642,E2 -24684.642} C_VEL
LIN {X 0,Y 153.927,Z 162.904,A -85,B 0,C 180,E1 -24687.049,E2 -24687.049} C_VEL
LIN {X 0,Y 155.684,Z 164.755,A -85,B 0,C 180,E1 -24688.674,E2 -24688.674} C_VEL
LIN {X 0,Y 158.427,Z 168.451,A -85,B 0,C 180,E1 -24691.047,E2 -24691.047} C_VEL
LIN {X 0,Y 162.776,Z 174.619,A -85,B 0,C 180,E1 -24694.351,E2 -24694.351} C_VEL
LIN {X 0,Y 167.605,Z 181.862,A -85,B 0,C 180,E1 -24697.54,E2 -24697.54} C_VEL
LIN {X 0,Y 173.425,Z 191.525,A -85,B 0,C 180,E1 -24700.924,E2 -24700.924} C_VEL
LIN {X 0,Y 178.347,Z 200.905,A -85,B 0,C 180,E1 -24703.513,E2 -24703.513} C_VEL
LIN {X 0,Y 181.252,Z 207.254,A -85,B 0,C 180,E1 -24704.963,E2 -24704.963} C_VEL
LIN {X 0,Y 176.876,Z 266.152,A -85,B 0,C 180,E1 -24706.947,E2 -24706.947} C_VEL
LIN {X 0,Y 174.944,Z 280.543,A -85,B 0,C 180,E1 -24707.807,E2 -24707.807} C_VEL
LIN {X 0,Y 172.163,Z 294.488,A -85,B 0,C 180,E1 -24709.028,E2 -24709.028} C_VEL
LIN {X 0,Y 168.755,Z 307.459,A -85,B 0,C 180,E1 -24710.573,E2 -24710.573} C_VEL
LIN {X 0,Y 164.681,Z 320.024,A -85,B 0,C 180,E1 -24712.545,E2 -24712.545} C_VEL
LIN {X 0,Y 160.471,Z 331.457,A -85,B 0,C 180,E1 -24714.913,E2 -24714.913} C_VEL
LIN {X 0,Y 155.578,Z 342.934,A -85,B 0,C 180,E1 -24717.942,E2 -24717.942} C_VEL
LIN {X 0,Y 150.683,Z 353.204,A -85,B 0,C 180,E1 -24721.441,E2 -24721.441} C_VEL
LIN {X 0,Y 146.398,Z 361.681,A -85,B 0,C 180,E1 -24725.163,E2 -24725.163} C_VEL
LIN {X 0,Y 142.227,Z 369.786,A -85,B 0,C 180,E1 -24729.764,E2 -24729.764} C_VEL
LIN {X 0,Y 139.204,Z 375.482,A -85,B 0,C 180,E1 -24733.879,E2 -24733.879} C_VEL
LIN {X 0,Y 136.751,Z 380.143,A -85,B 0,C 180,E1 -24738.138,E2 -24738.138} C_VEL
LIN {X 0,Y 135.208,Z 383.912,A -85,B 0,C 180,E1 -24742.534,E2 -24742.534} C_VEL
LIN {X 0,Y 134.052,Z 386.833,A -85,B 0,C 180,E1 -24746.995,E2 -24746.995} C_VEL
LIN {X 0,Y 133.423,Z 389.501,A -85,B 0,C 180,E1 -24753.02,E2 -24753.02} C_VEL
LIN {X 0,Y 133.299,Z 390.332,A -85,B 0,C 180,E1 -24756.053,E2 -24756.053} C_VEL
LIN {X 0,Y 133.557,Z 390.995,A -85,B 0,C 180,E1 -24762.151,E2 -24762.151} C_VEL
LIN {X 0,Y 134.918,Z 390.316,A -85,B 0,C 180,E1 -24768.213,E2 -24768.213} C_VEL
LIN {X 0,Y 137.403,Z 388.284,A -85,B 0,C 180,E1 -24774.154,E2 -24774.154} C_VEL
LIN {X 0,Y 141.097,Z 384.839,A -85,B 0,C 180,E1 -24779.875,E2 -24779.875} C_VEL
LIN {X 0,Y 146.034,Z 379.871,A -85,B 0,C 180,E1 -24785.276,E2 -24785.276} C_VEL
LIN {X 0,Y 150.509,Z 375.038,A -85,B 0,C 180,E1 -24789.079,E2 -24789.079} C_VEL
LIN {X 0,Y 156.496,Z 368.035,A -85,B 0,C 180,E1 -24793.224,E2 -24793.224} C_VEL
LIN {X 0,Y 163.096,Z 359.323,A -85,B 0,C 180,E1 -24797.101,E2 -24797.101} C_VEL
LIN {X 0,Y 169.394,Z 350.184,A -85,B 0,C 180,E1 -24800.134,E2 -24800.134} C_VEL
LIN {X 0,Y 176.183,Z 339.082,A -85,B 0,C 180,E1 -24802.922,E2 -24802.922} C_VEL
LIN {X 0,Y 181.994,Z 327.692,A -85,B 0,C 180,E1 -24805.146,E2 -24805.146} C_VEL
LIN {X 0,Y 187.014,Z 316.671,A -85,B 0,C 180,E1 -24806.737,E2 -24806.737} C_VEL
LIN {X 0,Y 191.667,Z 303.817,A -85,B 0,C 180,E1 -24808.238,E2 -24808.238} C_VEL
LIN {X 0,Y 195.47,Z 290.565,A -85,B 0,C 180,E1 -24809.391,E2 -24809.391} C_VEL
LIN {X 0,Y 198.29,Z 277.308,A -85,B 0,C 180,E1 -24810.236,E2 -24810.236} C_VEL
LIN {X 0,Y 200.396,Z 262.833,A -85,B 0,C 180,E1 -24810.809,E2 -24810.809} C_VEL
LIN {X 0,Y 203.483,Z 226.507,A -85,B 0,C 180,E1 -24811.843,E2 -24811.843} C_VEL
LIN {X 0,Y 200.769,Z 220.428,A -85,B 0,C 180,E1 -24813.579,E2 -24813.579} C_VEL
LIN {X 0,Y 195.899,Z 211.515,A -85,B 0,C 180,E1 -24816.931,E2 -24816.931} C_VEL
LIN {X 0,Y 191.881,Z 204.835,A -85,B 0,C 180,E1 -24820.126,E2 -24820.126} C_VEL
LIN {X 0,Y 189.602,Z 201.254,A -85,B 0,C 180,E1 -24822.193,E2 -24822.193} C_VEL
LIN {X 0,Y 187.474,Z 197.939,A -85,B 0,C 180,E1 -24824.368,E2 -24824.368} C_VEL
LIN {X 0,Y 184.992,Z 194.072,A -85,B 0,C 180,E1 -24827.347,E2 -24827.347} C_VEL
LIN {X 0,Y 182.63,Z 190.525,A -85,B 0,C 180,E1 -24830.918,E2 -24830.918} C_VEL
LIN {X 0,Y 182.164,Z 189.558,A -85,B 0,C 180,E1 -24831.821,E2 -24831.821} C_VEL
LIN {X 0,Y 179.759,Z 186.237,A -85,B 0,C 180,E1 -24838.284,E2 -24838.284} C_VEL
LIN {X 0,Y 179.518,Z 184.602,A -85,B 0,C 180,E1 -24840.634,E2 -24840.634} C_VEL
LIN {X 0,Y 179.529,Z 184.858,A -85,B 0,C 180,E1 -24845.41,E2 -24845.41} C_VEL
LIN {X 0,Y 180.824,Z 188.53,A -85,B 0,C 180,E1 -24851.205,E2 -24851.205} C_VEL
LIN {X 0,Y 182.371,Z 190.107,A -85,B 0,C 180,E1 -24854.342,E2 -24854.342} C_VEL
LIN {X 0,Y 184.652,Z 193.799,A -85,B 0,C 180,E1 -24857.959,E2 -24857.959} C_VEL
LIN {X 0,Y 185.569,Z 195.035,A -85,B 0,C 180,E1 -24859.137,E2 -24859.137} C_VEL
LIN {X 0,Y 188.478,Z 199.464,A -85,B 0,C 180,E1 -24862.418,E2 -24862.418} C_VEL
LIN {X 0,Y 190.646,Z 202.988,A -85,B 0,C 180,E1 -24864.521,E2 -24864.521} C_VEL
LIN {X 0,Y 194.267,Z 210.169,A -85,B 0,C 180,E1 -24867.681,E2 -24867.681} C_VEL
LIN {X 0,Y 198.679,Z 219.946,A -85,B 0,C 180,E1 -24871.027,E2 -24871.027} C_VEL
LIN {X 0,Y 202.398,Z 229.278,A -85,B 0,C 180,E1 -24873.563,E2 -24873.563} C_VEL
LIN {X 0,Y 203.134,Z 231.24,A -85,B 0,C 180,E1 -24874.04,E2 -24874.04} C_VEL
LIN {X 0,Y 199.686,Z 271.06,A -85,B 0,C 180,E1 -24875.183,E2 -24875.183} C_VEL
LIN {X 0,Y 197.205,Z 285.865,A -85,B 0,C 180,E1 -24875.829,E2 -24875.829} C_VEL
LIN {X 0,Y 193.916,Z 299.272,A -85,B 0,C 180,E1 -24876.691,E2 -24876.691} C_VEL
LIN {X 0,Y 189.403,Z 313.252,A -85,B 0,C 180,E1 -24877.954,E2 -24877.954} C_VEL
LIN {X 0,Y 184.405,Z 325.749,A -85,B 0,C 180,E1 -24879.487,E2 -24879.487} C_VEL
LIN {X 0,Y 178.907,Z 337.172,A -85,B 0,C 180,E1 -24881.298,E2 -24881.298} C_VEL
LIN {X 0,Y 173.711,Z 346.694,A -85,B 0,C 180,E1 -24883.26,E2 -24883.26} C_VEL
LIN {X 0,Y 167.146,Z 357.294,A -85,B 0,C 180,E1 -24886.07,E2 -24886.07} C_VEL
LIN {X 0,Y 160.967,Z 366.061,A -85,B 0,C 180,E1 -24889.086,E2 -24889.086} C_VEL
LIN {X 0,Y 155.285,Z 373.368,A -85,B 0,C 180,E1 -24892.338,E2 -24892.338} C_VEL
LIN {X 0,Y 150.008,Z 379.636,A -85,B 0,C 180,E1 -24895.939,E2 -24895.939} C_VEL
LIN {X 0,Y 144.246,Z 385.976,A -85,B 0,C 180,E1 -24900.841,E2 -24900.841} C_VEL
LIN {X 0,Y 142.616,Z 387.719,A -85,B 0,C 180,E1 -24902.538,E2 -24902.538} C_VEL
LIN {X 0,Y 140.284,Z 389.655,A -85,B 0,C 180,E1 -24904.6,E2 -24904.6} C_VEL
LIN {X 0,Y 134.959,Z 392.31,A -85,B 0,C 180,E1 -24907.907,E2 -24907.907} C_VEL
LIN {X 0,Y 130.824,Z 394.003,A -85,B 0,C 180,E1 -24910.751,E2 -24910.751} C_VEL
LIN {X 0,Y 128.679,Z 395.013,A -85,B 0,C 180,E1 -24913.143,E2 -24913.143} C_VEL
LIN {X 0,Y 128.277,Z 395.325,A -85,B 0,C 180,E1 -24913.992,E2 -24913.992} C_VEL
LIN {X 0,Y 126.68,Z 396.713,A -85,B 0,C 180,E1 -24920.419,E2 -24920.419} C_VEL
LIN {X 0,Y 126.3,Z 396.738,A -85,B 0,C 180,E1 -24926.81,E2 -24926.81} C_VEL
LIN {X 0,Y 126.388,Z 396.249,A -85,B 0,C 180,E1 -24929.999,E2 -24929.999} C_VEL
LIN {X 0,Y 126.3,Z 395.411,A -85,B 0,C 180,E1 -24933.189,E2 -24933.189} C_VEL
LIN {X 0,Y 126.651,Z 392.685,A -85,B 0,C 180,E1 -24939.582,E2 -24939.582} C_VEL
LIN {X 0,Y 128.027,Z 388.493,A -85,B 0,C 180,E1 -24945.93,E2 -24945.93} C_VEL
LIN {X 0,Y 130.809,Z 382.719,A -85,B 0,C 180,E1 -24952.091,E2 -24952.091} C_VEL
LIN {X 0,Y 133.689,Z 377.067,A -85,B 0,C 180,E1 -24956.661,E2 -24956.661} C_VEL
LIN {X 0,Y 137.946,Z 369.336,A -85,B 0,C 180,E1 -24961.48,E2 -24961.48} C_VEL
LIN {X 0,Y 142.329,Z 361.097,A -85,B 0,C 180,E1 -24965.464,E2 -24965.464} C_VEL
LIN {X 0,Y 147.525,Z 351.175,A -85,B 0,C 180,E1 -24969.14,E2 -24969.14} C_VEL
LIN {X 0,Y 152.078,Z 341.566,A -85,B 0,C 180,E1 -24971.928,E2 -24971.928} C_VEL
LIN {X 0,Y 156.663,Z 330.458,A -85,B 0,C 180,E1 -24974.502,E2 -24974.502} C_VEL
LIN {X 0,Y 160.908,Z 318.881,A -85,B 0,C 180,E1 -24976.562,E2 -24976.562} C_VEL
LIN {X 0,Y 164.86,Z 306.305,A -85,B 0,C 180,E1 -24978.247,E2 -24978.247} C_VEL
LIN {X 0,Y 168.331,Z 292.29,A -85,B 0,C 180,E1 -24979.636,E2 -24979.636} C_VEL
LIN {X 0,Y 170.827,Z 278.434,A -85,B 0,C 180,E1 -24980.594,E2 -24980.594} C_VEL
LIN {X 0,Y 172.482,Z 263.98,A -85,B 0,C 180,E1 -24981.205,E2 -24981.205} C_VEL
LIN {X 0,Y 176.081,Z 214.308,A -85,B 0,C 180,E1 -24982.906,E2 -24982.906} C_VEL
LIN {X 0,Y 172.465,Z 204.197,A -85,B 0,C 180,E1 -24985.019,E2 -24985.019} C_VEL
LIN {X 0,Y 167.823,Z 193.211,A -85,B 0,C 180,E1 -24987.89,E2 -24987.89} C_VEL
LIN {X 0,Y 165.535,Z 188.746,A -85,B 0,C 180,E1 -24989.372,E2 -24989.372} C_VEL
LIN {X 0,Y 161.135,Z 181.891,A -85,B 0,C 180,E1 -24992.379,E2 -24992.379} C_VEL
LIN {X 0,Y 158.131,Z 177.491,A -85,B 0,C 180,E1 -24994.674,E2 -24994.674} C_VEL
LIN {X 0,Y 156.028,Z 174.494,A -85,B 0,C 180,E1 -24996.437,E2 -24996.437} C_VEL
LIN {X 0,Y 153.001,Z 170.272,A -85,B 0,C 180,E1 -24999.271,E2 -24999.271} C_VEL
LIN {X 0,Y 150.307,Z 166.744,A -85,B 0,C 180,E1 -25002.175,E2 -25002.175} C_VEL
LIN {X 0,Y 149.669,Z 165.613,A -85,B 0,C 180,E1 -25002.978,E2 -25002.978} C_VEL
LIN {X 0,Y 147.087,Z 162.995,A -85,B 0,C 180,E1 -25006.355,E2 -25006.355} C_VEL
LIN {X 0,Y 145.914,Z 160.456,A -85,B 0,C 180,E1 -25008.431,E2 -25008.431} C_VEL
LIN {X 0,Y 142.709,Z 157.575,A -85,B 0,C 180,E1 -25015.632,E2 -25015.632} C_VEL
LIN {X 0,Y 142.093,Z 155.17,A -85,B 0,C 180,E1 -25019.336,E2 -25019.336} C_VEL
LIN {X 0,Y 142.053,Z 154.684,A -85,B 0,C 180,E1 -25020.001,E2 -25020.001} C_VEL
LIN {X 0,Y 141.863,Z 155.013,A -85,B 0,C 180,E1 -25024.974,E2 -25024.974} C_VEL
LIN {X 0,Y 144.349,Z 159.713,A -85,B 0,C 180,E1 -25035.174,E2 -25035.174} C_VEL
LIN {X 0,Y 145.953,Z 160.779,A -85,B 0,C 180,E1 -25038.059,E2 -25038.059} C_VEL
LIN {X 0,Y 147.513,Z 163.742,A -85,B 0,C 180,E1 -25040.677,E2 -25040.677} C_VEL
LIN {X 0,Y 149.982,Z 166.148,A -85,B 0,C 180,E1 -25043.793,E2 -25043.793} C_VEL
LIN {X 0,Y 152.389,Z 169.726,A -85,B 0,C 180,E1 -25046.512,E2 -25046.512} C_VEL
LIN {X 0,Y 153.676,Z 171.187,A -85,B 0,C 180,E1 -25047.769,E2 -25047.769} C_VEL
LIN {X 0,Y 157.318,Z 176.373,A -85,B 0,C 180,E1 -25051.041,E2 -25051.041} C_VEL
LIN {X 0,Y 160.553,Z 181.114,A -85,B 0,C 180,E1 -25053.578,E2 -25053.578} C_VEL
LIN {X 0,Y 165.434,Z 188.793,A -85,B 0,C 180,E1 -25056.955,E2 -25056.955} C_VEL
LIN {X 0,Y 170.519,Z 197.627,A -85,B 0,C 180,E1 -25060.059,E2 -25060.059} C_VEL
LIN {X 0,Y 175.36,Z 207.34,A -85,B 0,C 180,E1 -25062.75,E2 -25062.75} C_VEL
LIN {X 0,Y 176.387,Z 209.536,A -85,B 0,C 180,E1 -25063.292,E2 -25063.292} C_VEL
LIN {X 0,Y 172.066,Z 266.282,A -85,B 0,C 180,E1 -25065.243,E2 -25065.243} C_VEL
LIN {X 0,Y 170.068,Z 280.562,A -85,B 0,C 180,E1 -25066.094,E2 -25066.094} C_VEL
LIN {X 0,Y 167.171,Z 294.545,A -85,B 0,C 180,E1 -25067.32,E2 -25067.32} C_VEL
LIN {X 0,Y 163.919,Z 306.656,A -85,B 0,C 180,E1 -25068.762,E2 -25068.762} C_VEL
LIN {X 0,Y 159.661,Z 319.409,A -85,B 0,C 180,E1 -25070.747,E2 -25070.747} C_VEL
LIN {X 0,Y 155.243,Z 330.98,A -85,B 0,C 180,E1 -25073.142,E2 -25073.142} C_VEL
LIN {X 0,Y 150.551,Z 341.595,A -85,B 0,C 180,E1 -25075.932,E2 -25075.932} C_VEL
LIN {X 0,Y 145.359,Z 352.118,A -85,B 0,C 180,E1 -25079.492,E2 -25079.492} C_VEL
LIN {X 0,Y 140.697,Z 360.807,A -85,B 0,C 180,E1 -25083.285,E2 -25083.285} C_VEL
LIN {X 0,Y 136.192,Z 369.136,A -85,B 0,C 180,E1 -25088.03,E2 -25088.03} C_VEL
LIN {X 0,Y 132.415,Z 375.848,A -85,B 0,C 180,E1 -25093.028,E2 -25093.028} C_VEL
LIN {X 0,Y 129.842,Z 380.466,A -85,B 0,C 180,E1 -25097.496,E2 -25097.496} C_VEL
LIN {X 0,Y 127.661,Z 385.258,A -85,B 0,C 180,E1 -25103.679,E2 -25103.679} C_VEL
LIN {X 0,Y 126.546,Z 388.582,A -85,B 0,C 180,E1 -25110.001,E2 -25110.001} C_VEL
LIN {X 0,Y 126.309,Z 389.724,A -85,B 0,C 180,E1 -25113.19,E2 -25113.19} C_VEL
LIN {X 0,Y 126.195,Z 390.532,A -85,B 0,C 180,E1 -25116.396,E2 -25116.396} C_VEL
LIN {X 0,Y 126.531,Z 391.152,A -85,B 0,C 180,E1 -25122.837,E2 -25122.837} C_VEL
LIN {X 0,Y 128.081,Z 390.436,A -85,B 0,C 180,E1 -25129.223,E2 -25129.223} C_VEL
LIN {X 0,Y 130.827,Z 388.366,A -85,B 0,C 180,E1 -25135.453,E2 -25135.453} C_VEL
LIN {X 0,Y 134.879,Z 384.882,A -85,B 0,C 180,E1 -25141.404,E2 -25141.404} C_VEL
LIN {X 0,Y 140.2,Z 379.873,A -85,B 0,C 180,E1 -25146.981,E2 -25146.981} C_VEL
LIN {X 0,Y 144.97,Z 374.996,A -85,B 0,C 180,E1 -25150.88,E2 -25150.88} C_VEL
LIN {X 0,Y 151.261,Z 367.968,A -85,B 0,C 180,E1 -25155.097,E2 -25155.097} C_VEL
LIN {X 0,Y 158.256,Z 359.177,A -85,B 0,C 180,E1 -25159.022,E2 -25159.022} C_VEL
LIN {X 0,Y 164.854,Z 349.975,A -85,B 0,C 180,E1 -25162.064,E2 -25162.064} C_VEL
LIN {X 0,Y 171.333,Z 339.792,A -85,B 0,C 180,E1 -25164.614,E2 -25164.614} C_VEL
LIN {X 0,Y 177.363,Z 328.559,A -85,B 0,C 180,E1 -25166.833,E2 -25166.833} C_VEL
LIN {X 0,Y 183.156,Z 316.113,A -85,B 0,C 180,E1 -25168.625,E2 -25168.625} C_VEL
LIN {X 0,Y 187.66,Z 304.081,A -85,B 0,C 180,E1 -25170.003,E2 -25170.003} C_VEL
LIN {X 0,Y 191.576,Z 290.86,A -85,B 0,C 180,E1 -25171.147,E2 -25171.147} C_VEL
LIN {X 0,Y 194.533,Z 277.448,A -85,B 0,C 180,E1 -25171.987,E2 -25171.987} C_VEL
LIN {X 0,Y 196.685,Z 263.009,A -85,B 0,C 180,E1 -25172.556,E2 -25172.556} C_VEL
LIN {X 0,Y 199.602,Z 229.481,A -85,B 0,C 180,E1 -25173.522,E2 -25173.522} C_VEL
LIN {X 0,Y 196.739,Z 223.421,A -85,B 0,C 180,E1 -25175.498,E2 -25175.498} C_VEL
LIN {X 0,Y 192.56,Z 215.534,A -85,B 0,C 180,E1 -25178.681,E2 -25178.681} C_VEL
LIN {X 0,Y 188.44,Z 208.508,A -85,B 0,C 180,E1 -25182.36,E2 -25182.36} C_VEL
LIN {X 0,Y 185.783,Z 204.373,A -85,B 0,C 180,E1 -25185.17,E2 -25185.17} C_VEL
LIN {X 0,Y 183.481,Z 200.64,A -85,B 0,C 180,E1 -25188.118,E2 -25188.118} C_VEL
LIN {X 0,Y 181.305,Z 197.05,A -85,B 0,C 180,E1 -25191.694,E2 -25191.694} C_VEL
LIN {X 0,Y 180.922,Z 196.378,A -85,B 0,C 180,E1 -25192.466,E2 -25192.466} C_VEL
LIN {X 0,Y 178.724,Z 192.79,A -85,B 0,C 180,E1 -25199.296,E2 -25199.296} C_VEL
LIN {X 0,Y 178.639,Z 191.743,A -85,B 0,C 180,E1 -25200.637,E2 -25200.637} C_VEL
LIN {X 0,Y 178.578,Z 191.742,A -85,B 0,C 180,E1 -25204.514,E2 -25204.514} C_VEL
LIN {X 0,Y 178.818,Z 193.244,A -85,B 0,C 180,E1 -25207.125,E2 -25207.125} C_VEL
LIN {X 0,Y 180.263,Z 195.952,A -85,B 0,C 180,E1 -25211.952,E2 -25211.952} C_VEL
LIN {X 0,Y 181.157,Z 196.874,A -85,B 0,C 180,E1 -25213.76,E2 -25213.76} C_VEL
LIN {X 0,Y 183.437,Z 200.65,A -85,B 0,C 180,E1 -25217.56,E2 -25217.56} C_VEL
LIN {X 0,Y 186.662,Z 205.692,A -85,B 0,C 180,E1 -25221.536,E2 -25221.536} C_VEL
LIN {X 0,Y 188.812,Z 209.433,A -85,B 0,C 180,E1 -25223.763,E2 -25223.763} C_VEL
LIN {X 0,Y 192.094,Z 216.343,A -85,B 0,C 180,E1 -25226.811,E2 -25226.811} C_VEL
LIN {X 0,Y 195.933,Z 225.273,A -85,B 0,C 180,E1 -25229.921,E2 -25229.921} C_VEL
LIN {X 0,Y 199.224,Z 233.913,A -85,B 0,C 180,E1 -25232.332,E2 -25232.332} C_VEL
LIN {X 0,Y 195.906,Z 271.506,A -85,B 0,C 180,E1 -25233.454,E2 -25233.454} C_VEL
LIN {X 0,Y 193.332,Z 286.164,A -85,B 0,C 180,E1 -25234.091,E2 -25234.091} C_VEL
LIN {X 0,Y 189.786,Z 300.013,A -85,B 0,C 180,E1 -25234.983,E2 -25234.983} C_VEL
LIN {X 0,Y 185.148,Z 313.794,A -85,B 0,C 180,E1 -25236.232,E2 -25236.232} C_VEL
LIN {X 0,Y 179.995,Z 326.155,A -85,B 0,C 180,E1 -25237.751,E2 -25237.751} C_VEL
LIN {X 0,Y 174.306,Z 337.478,A -85,B 0,C 180,E1 -25239.545,E2 -25239.545} C_VEL
LIN {X 0,Y 168.25,Z 348.049,A -85,B 0,C 180,E1 -25241.77,E2 -25241.77} C_VEL
LIN {X 0,Y 162.092,Z 357.456,A -85,B 0,C 180,E1 -25244.323,E2 -25244.323} C_VEL
LIN {X 0,Y 155.67,Z 366.168,A -85,B 0,C 180,E1 -25247.374,E2 -25247.374} C_VEL
LIN {X 0,Y 149.705,Z 373.428,A -85,B 0,C 180,E1 -25250.671,E2 -25250.671} C_VEL
LIN {X 0,Y 144.315,Z 379.489,A -85,B 0,C 180,E1 -25254.24,E2 -25254.24} C_VEL
LIN {X 0,Y 138.063,Z 385.955,A -85,B 0,C 180,E1 -25259.4,E2 -25259.4} C_VEL
LIN {X 0,Y 133.213,Z 390.805,A -85,B 0,C 180,E1 -25265.035,E2 -25265.035} C_VEL
LIN {X 0,Y 129.525,Z 394.189,A -85,B 0,C 180,E1 -25271,E2 -25271} C_VEL
LIN {X 0,Y 128.277,Z 395.325,A -85,B 0,C 180,E1 -25273.992,E2 -25273.992} C_VEL
LIN {X 0,Y 126.826,Z 396.124,A -85,B 0,C 180,E1 -25276.537,E2 -25276.537} C_VEL
LIN {X 0,Y 123.135,Z 396.763,A -85,B 0,C 180,E1 -25280.745,E2 -25280.745} C_VEL
LIN {X 0,Y 120.385,Z 396.744,A -85,B 0,C 180,E1 -25284.281,E2 -25284.281} C_VEL
LIN {X 0,Y 119.273,Z 396.491,A -85,B 0,C 180,E1 -25287.08,E2 -25287.08} C_VEL
LIN {X 0,Y 119.196,Z 396.341,A -85,B 0,C 180,E1 -25288.033,E2 -25288.033} C_VEL
LIN {X 0,Y 119.29,Z 396.047,A -85,B 0,C 180,E1 -25289.999,E2 -25289.999} C_VEL
LIN {X 0,Y 119.194,Z 395.191,A -85,B 0,C 180,E1 -25293.38,E2 -25293.38} C_VEL
LIN {X 0,Y 119.628,Z 392.432,A -85,B 0,C 180,E1 -25300.151,E2 -25300.151} C_VEL
LIN {X 0,Y 121.165,Z 388.204,A -85,B 0,C 180,E1 -25306.858,E2 -25306.858} C_VEL
LIN {X 0,Y 124.194,Z 382.392,A -85,B 0,C 180,E1 -25313.335,E2 -25313.335} C_VEL
LIN {X 0,Y 127.727,Z 376.028,A -85,B 0,C 180,E1 -25318.602,E2 -25318.602} C_VEL
LIN {X 0,Y 131.88,Z 368.923,A -85,B 0,C 180,E1 -25323.108,E2 -25323.108} C_VEL
LIN {X 0,Y 136.547,Z 360.632,A -85,B 0,C 180,E1 -25327.211,E2 -25327.211} C_VEL
LIN {X 0,Y 142.058,Z 350.654,A -85,B 0,C 180,E1 -25330.958,E2 -25330.958} C_VEL
LIN {X 0,Y 147.191,Z 340.217,A -85,B 0,C 180,E1 -25333.992,E2 -25333.992} C_VEL
LIN {X 0,Y 152.165,Z 328.469,A -85,B 0,C 180,E1 -25336.672,E2 -25336.672} C_VEL
LIN {X 0,Y 156.664,Z 316.487,A -85,B 0,C 180,E1 -25338.712,E2 -25338.712} C_VEL
LIN {X 0,Y 160.79,Z 303.285,A -85,B 0,C 180,E1 -25340.387,E2 -25340.387} C_VEL
LIN {X 0,Y 164.275,Z 288.812,A -85,B 0,C 180,E1 -25341.7,E2 -25341.7} C_VEL
LIN {X 0,Y 166.541,Z 275.417,A -85,B 0,C 180,E1 -25342.549,E2 -25342.549} C_VEL
LIN {X 0,Y 168.323,Z 257.583,A -85,B 0,C 180,E1 -25343.231,E2 -25343.231} C_VEL
LIN {X 0,Y 171.408,Z 216.505,A -85,B 0,C 180,E1 -25344.652,E2 -25344.652} C_VEL
LIN {X 0,Y 168.141,Z 207.215,A -85,B 0,C 180,E1 -25346.733,E2 -25346.733} C_VEL
LIN {X 0,Y 164.128,Z 197.426,A -85,B 0,C 180,E1 -25349.437,E2 -25349.437} C_VEL
LIN {X 0,Y 162.135,Z 193.569,A -85,B 0,C 180,E1 -25350.825,E2 -25350.825} C_VEL
LIN {X 0,Y 158.123,Z 187.141,A -85,B 0,C 180,E1 -25353.789,E2 -25353.789} C_VEL
LIN {X 0,Y 154.146,Z 181.017,A -85,B 0,C 180,E1 -25357.177,E2 -25357.177} C_VEL
LIN {X 0,Y 151.158,Z 176.777,A -85,B 0,C 180,E1 -25360.117,E2 -25360.117} C_VEL
LIN {X 0,Y 148.435,Z 172.975,A -85,B 0,C 180,E1 -25363.264,E2 -25363.264} C_VEL
LIN {X 0,Y 147.633,Z 171.971,A -85,B 0,C 180,E1 -25364.291,E2 -25364.291} C_VEL
LIN {X 0,Y 145.325,Z 169.088,A -85,B 0,C 180,E1 -25367.686,E2 -25367.686} C_VEL
LIN {X 0,Y 144.575,Z 167.307,A -85,B 0,C 180,E1 -25369.156,E2 -25369.156} C_VEL
LIN {X 0,Y 141.472,Z 163.959,A -85,B 0,C 180,E1 -25377.153,E2 -25377.153} C_VEL
LIN {X 0,Y 141.139,Z 161.731,A -85,B 0,C 180,E1 -25380.357,E2 -25380.357} C_VEL
LIN {X 0,Y 140.984,Z 162.127,A -85,B 0,C 180,E1 -25384.934,E2 -25384.934} C_VEL
LIN {X 0,Y 143.019,Z 166.452,A -85,B 0,C 180,E1 -25394.224,E2 -25394.224} C_VEL
LIN {X 0,Y 144.599,Z 167.636,A -85,B 0,C 180,E1 -25397.32,E2 -25397.32} C_VEL
LIN {X 0,Y 146.504,Z 170.961,A -85,B 0,C 180,E1 -25400.579,E2 -25400.579} C_VEL
LIN {X 0,Y 148.349,Z 172.888,A -85,B 0,C 180,E1 -25403.007,E2 -25403.007} C_VEL
LIN {X 0,Y 150.967,Z 176.609,A -85,B 0,C 180,E1 -25406.065,E2 -25406.065} C_VEL
LIN {X 0,Y 154.832,Z 182.152,A -85,B 0,C 180,E1 -25409.832,E2 -25409.832} C_VEL
LIN {X 0,Y 158.281,Z 187.44,A -85,B 0,C 180,E1 -25412.715,E2 -25412.715} C_VEL
LIN {X 0,Y 162.963,Z 195.115,A -85,B 0,C 180,E1 -25416.133,E2 -25416.133} C_VEL
LIN {X 0,Y 167.907,Z 204.192,A -85,B 0,C 180,E1 -25419.318,E2 -25419.318} C_VEL
LIN {X 0,Y 171.719,Z 212.326,A -85,B 0,C 180,E1 -25421.578,E2 -25421.578} C_VEL
LIN {X 0,Y 167.425,Z 266.327,A -85,B 0,C 180,E1 -25423.438,E2 -25423.438} C_VEL
LIN {X 0,Y 165.352,Z 280.58,A -85,B 0,C 180,E1 -25424.283,E2 -25424.283} C_VEL
LIN {X 0,Y 162.354,Z 294.598,A -85,B 0,C 180,E1 -25425.515,E2 -25425.515} C_VEL
LIN {X 0,Y 158.677,Z 307.614,A -85,B 0,C 180,E1 -25427.081,E2 -25427.081} C_VEL
LIN {X 0,Y 154.27,Z 320.211,A -85,B 0,C 180,E1 -25429.091,E2 -25429.091} C_VEL
LIN {X 0,Y 149.659,Z 331.669,A -85,B 0,C 180,E1 -25431.522,E2 -25431.522} C_VEL
LIN {X 0,Y 144.744,Z 342.197,A -85,B 0,C 180,E1 -25434.363,E2 -25434.363} C_VEL
LIN {X 0,Y 139.309,Z 352.647,A -85,B 0,C 180,E1 -25438.014,E2 -25438.014} C_VEL
LIN {X 0,Y 134.417,Z 361.275,A -85,B 0,C 180,E1 -25441.93,E2 -25441.93} C_VEL
LIN {X 0,Y 129.653,Z 369.548,A -85,B 0,C 180,E1 -25446.86,E2 -25446.86} C_VEL
LIN {X 0,Y 125.668,Z 376.205,A -85,B 0,C 180,E1 -25452.087,E2 -25452.087} C_VEL
LIN {X 0,Y 122.322,Z 382.118,A -85,B 0,C 180,E1 -25458.4,E2 -25458.4} C_VEL
LIN {X 0,Y 120.619,Z 385.541,A -85,B 0,C 180,E1 -25463.309,E2 -25463.309} C_VEL
LIN {X 0,Y 119.441,Z 388.822,A -85,B 0,C 180,E1 -25470.001,E2 -25470.001} C_VEL
LIN {X 0,Y 119.188,Z 389.941,A -85,B 0,C 180,E1 -25473.381,E2 -25473.381} C_VEL
LIN {X 0,Y 119.094,Z 390.726,A -85,B 0,C 180,E1 -25476.779,E2 -25476.779} C_VEL
LIN {X 0,Y 119.528,Z 391.308,A -85,B 0,C 180,E1 -25483.603,E2 -25483.603} C_VEL
LIN {X 0,Y 121.295,Z 390.555,A -85,B 0,C 180,E1 -25490.344,E2 -25490.344} C_VEL
LIN {X 0,Y 124.329,Z 388.448,A -85,B 0,C 180,E1 -25496.887,E2 -25496.887} C_VEL
LIN {X 0,Y 128.765,Z 384.925,A -85,B 0,C 180,E1 -25503.08,E2 -25503.08} C_VEL
LIN {X 0,Y 134.507,Z 379.875,A -85,B 0,C 180,E1 -25508.83,E2 -25508.83} C_VEL
LIN {X 0,Y 139.586,Z 374.953,A -85,B 0,C 180,E1 -25512.822,E2 -25512.822} C_VEL
LIN {X 0,Y 146.181,Z 367.951,A -85,B 0,C 180,E1 -25517.065,E2 -25517.065} C_VEL
LIN {X 0,Y 152.53,Z 360.397,A -85,B 0,C 180,E1 -25520.514,E2 -25520.514} C_VEL
LIN {X 0,Y 159.348,Z 351.41,A -85,B 0,C 180,E1 -25523.602,E2 -25523.602} C_VEL
LIN {X 0,Y 165.417,Z 342.465,A -85,B 0,C 180,E1 -25525.944,E2 -25525.944} C_VEL
LIN {X 0,Y 171.64,Z 331.669,A -85,B 0,C 180,E1 -25528.212,E2 -25528.212} C_VEL
LIN {X 0,Y 177.515,Z 320.05,A -85,B 0,C 180,E1 -25530.004,E2 -25530.004} C_VEL
LIN {X 0,Y 182.814,Z 307.128,A -85,B 0,C 180,E1 -25531.57,E2 -25531.57} C_VEL
LIN {X 0,Y 187.202,Z 293.656,A -85,B 0,C 180,E1 -25532.784,E2 -25532.784} C_VEL
LIN {X 0,Y 190.573,Z 279.788,A -85,B 0,C 180,E1 -25533.689,E2 -25533.689} C_VEL
LIN {X 0,Y 192.85,Z 266.178,A -85,B 0,C 180,E1 -25534.267,E2 -25534.267} C_VEL
LIN {X 0,Y 195.916,Z 232.713,A -85,B 0,C 180,E1 -25535.238,E2 -25535.238} C_VEL
LIN {X 0,Y 191.699,Z 224.042,A -85,B 0,C 180,E1 -25538.492,E2 -25538.492} C_VEL
LIN {X 0,Y 187.896,Z 217.154,A -85,B 0,C 180,E1 -25541.885,E2 -25541.885} C_VEL
LIN {X 0,Y 185.766,Z 213.538,A -85,B 0,C 180,E1 -25544.08,E2 -25544.08} C_VEL
LIN {X 0,Y 183.97,Z 210.531,A -85,B 0,C 180,E1 -25546.186,E2 -25546.186} C_VEL
LIN {X 0,Y 182.033,Z 207.199,A -85,B 0,C 180,E1 -25548.869,E2 -25548.869} C_VEL
LIN {X 0,Y 180.036,Z 203.639,A -85,B 0,C 180,E1 -25552.429,E2 -25552.429} C_VEL
LIN {X 0,Y 177.773,Z 199.504,A -85,B 0,C 180,E1 -25560,E2 -25560} C_VEL
LIN {X 0,Y 177.724,Z 198.63,A -85,B 0,C 180,E1 -25561.28,E2 -25561.28} C_VEL
LIN {X 0,Y 177.728,Z 198.921,A -85,B 0,C 180,E1 -25564.845,E2 -25564.845} C_VEL
LIN {X 0,Y 178.951,Z 202.625,A -85,B 0,C 180,E1 -25570.937,E2 -25570.937} C_VEL
LIN {X 0,Y 180.064,Z 203.881,A -85,B 0,C 180,E1 -25573.399,E2 -25573.399} C_VEL
LIN {X 0,Y 182.193,Z 207.484,A -85,B 0,C 180,E1 -25577.105,E2 -25577.105} C_VEL
LIN {X 0,Y 185.244,Z 212.566,A -85,B 0,C 180,E1 -25581.053,E2 -25581.053} C_VEL
LIN {X 0,Y 186.988,Z 215.781,A -85,B 0,C 180,E1 -25582.96,E2 -25582.96} C_VEL
LIN {X 0,Y 190.057,Z 222.648,A -85,B 0,C 180,E1 -25585.995,E2 -25585.995} C_VEL
LIN {X 0,Y 193.589,Z 231.45,A -85,B 0,C 180,E1 -25589.05,E2 -25589.05} C_VEL
LIN {X 0,Y 195.592,Z 236.943,A -85,B 0,C 180,E1 -25590.637,E2 -25590.637} C_VEL
LIN {X 0,Y 192.376,Z 271.49,A -85,B 0,C 180,E1 -25591.643,E2 -25591.643} C_VEL
LIN {X 0,Y 189.823,Z 285.714,A -85,B 0,C 180,E1 -25592.245,E2 -25592.245} C_VEL
LIN {X 0,Y 186.176,Z 299.637,A -85,B 0,C 180,E1 -25593.116,E2 -25593.116} C_VEL
LIN {X 0,Y 181.738,Z 312.587,A -85,B 0,C 180,E1 -25594.249,E2 -25594.249} C_VEL
LIN {X 0,Y 176.388,Z 325.151,A -85,B 0,C 180,E1 -25595.725,E2 -25595.725} C_VEL
LIN {X 0,Y 170.538,Z 336.618,A -85,B 0,C 180,E1 -25597.504,E2 -25597.504} C_VEL
LIN {X 0,Y 164.313,Z 347.151,A -85,B 0,C 180,E1 -25599.655,E2 -25599.655} C_VEL
LIN {X 0,Y 157.2,Z 357.621,A -85,B 0,C 180,E1 -25602.466,E2 -25602.466} C_VEL
LIN {X 0,Y 150.52,Z 366.276,A -85,B 0,C 180,E1 -25605.543,E2 -25605.543} C_VEL
LIN {X 0,Y 143.29,Z 374.601,A -85,B 0,C 180,E1 -25609.467,E2 -25609.467} C_VEL
LIN {X 0,Y 136.831,Z 381.31,A -85,B 0,C 180,E1 -25613.795,E2 -25613.795} C_VEL
LIN {X 0,Y 130.504,Z 387.287,A -85,B 0,C 180,E1 -25619.231,E2 -25619.231} C_VEL
LIN {X 0,Y 126.782,Z 390.748,A -85,B 0,C 180,E1 -25623.674,E2 -25623.674} C_VEL
LIN {X 0,Y 122.808,Z 394.097,A -85,B 0,C 180,E1 -25629.917,E2 -25629.917} C_VEL
LIN {X 0,Y 120.37,Z 396.074,A -85,B 0,C 180,E1 -25636.493,E2 -25636.493} C_VEL
LIN {X 0,Y 119.305,Z 396.724,A -85,B 0,C 180,E1 -25643.233,E2 -25643.233} C_VEL
LIN {X 0,Y 119.196,Z 396.341,A -85,B 0,C 180,E1 -25648.033,E2 -25648.033} C_VEL
LIN {X 0,Y 118.891,Z 396.056,A -85,B 0,C 180,E1 -25649.909,E2 -25649.909} C_VEL
LIN {X 0,Y 118.082,Z 395.601,A -85,B 0,C 180,E1 -25651.76,E2 -25651.76} C_VEL
LIN {X 0,Y 115.721,Z 394.449,A -85,B 0,C 180,E1 -25655.439,E2 -25655.439} C_VEL
LIN {X 0,Y 113.525,Z 392.919,A -85,B 0,C 180,E1 -25659.241,E2 -25659.241} C_VEL
LIN {X 0,Y 112.9,Z 391.479,A -85,B 0,C 180,E1 -25662.175,E2 -25662.175} C_VEL
LIN {X 0,Y 113.015,Z 390.898,A -85,B 0,C 180,E1 -25663.155,E2 -25663.155} C_VEL
LIN {X 0,Y 115.052,Z 386.639,A -85,B 0,C 180,E1 -25669.631,E2 -25669.631} C_VEL
LIN {X 0,Y 117.65,Z 382.066,A -85,B 0,C 180,E1 -25674.718,E2 -25674.718} C_VEL
LIN {X 0,Y 121.598,Z 375.491,A -85,B 0,C 180,E1 -25680.349,E2 -25680.349} C_VEL
LIN {X 0,Y 126.708,Z 367.258,A -85,B 0,C 180,E1 -25685.618,E2 -25685.618} C_VEL
LIN {X 0,Y 131.833,Z 358.662,A -85,B 0,C 180,E1 -25689.77,E2 -25689.77} C_VEL
LIN {X 0,Y 137.726,Z 348.253,A -85,B 0,C 180,E1 -25693.541,E2 -25693.541} C_VEL
LIN {X 0,Y 142.969,Z 337.675,A -85,B 0,C 180,E1 -25696.512,E2 -25696.512} C_VEL
LIN {X 0,Y 147.912,Z 326.352,A -85,B 0,C 180,E1 -25698.963,E2 -25698.963} C_VEL
LIN {X 0,Y 152.673,Z 313.88,A -85,B 0,C 180,E1 -25700.968,E2 -25700.968} C_VEL
LIN {X 0,Y 156.957,Z 299.93,A -85,B 0,C 180,E1 -25702.634,E2 -25702.634} C_VEL
LIN {X 0,Y 160.245,Z 285.871,A -85,B 0,C 180,E1 -25703.828,E2 -25703.828} C_VEL
LIN {X 0,Y 162.463,Z 272.258,A -85,B 0,C 180,E1 -25704.602,E2 -25704.602} C_VEL
LIN {X 0,Y 165.08,Z 242.428,A -85,B 0,C 180,E1 -25705.655,E2 -25705.655} C_VEL
LIN {X 0,Y 166.916,Z 218.649,A -85,B 0,C 180,E1 -25706.491,E2 -25706.491} C_VEL
LIN {X 0,Y 163.225,Z 208.266,A -85,B 0,C 180,E1 -25709.07,E2 -25709.07} C_VEL
LIN {X 0,Y 159.959,Z 200.314,A -85,B 0,C 180,E1 -25711.511,E2 -25711.511} C_VEL
LIN {X 0,Y 155.56,Z 192.915,A -85,B 0,C 180,E1 -25714.958,E2 -25714.958} C_VEL
LIN {X 0,Y 152.026,Z 187.251,A -85,B 0,C 180,E1 -25718.178,E2 -25718.178} C_VEL
LIN {X 0,Y 149.089,Z 182.989,A -85,B 0,C 180,E1 -25721.269,E2 -25721.269} C_VEL
LIN {X 0,Y 146.326,Z 178.846,A -85,B 0,C 180,E1 -25724.772,E2 -25724.772} C_VEL
LIN {X 0,Y 143.866,Z 175.621,A -85,B 0,C 180,E1 -25728.615,E2 -25728.615} C_VEL
LIN {X 0,Y 143.087,Z 174.02,A -85,B 0,C 180,E1 -25730.22,E2 -25730.22} C_VEL
LIN {X 0,Y 140.49,Z 170.866,A -85,B 0,C 180,E1 -25737.671,E2 -25737.671} C_VEL
LIN {X 0,Y 140.221,Z 168.853,A -85,B 0,C 180,E1 -25740.718,E2 -25740.718} C_VEL
LIN {X 0,Y 140.099,Z 169.019,A -85,B 0,C 180,E1 -25744.316,E2 -25744.316} C_VEL
LIN {X 0,Y 141.993,Z 173.433,A -85,B 0,C 180,E1 -25753.904,E2 -25753.904} C_VEL
LIN {X 0,Y 143.317,Z 174.522,A -85,B 0,C 180,E1 -25756.654,E2 -25756.654} C_VEL
LIN {X 0,Y 145.254,Z 177.869,A -85,B 0,C 180,E1 -25760.119,E2 -25760.119} C_VEL
LIN {X 0,Y 146.8,Z 179.647,A -85,B 0,C 180,E1 -25762.27,E2 -25762.27} C_VEL
LIN {X 0,Y 150.003,Z 184.333,A -85,B 0,C 180,E1 -25766.125,E2 -25766.125} C_VEL
LIN {X 0,Y 153.27,Z 189.356,A -85,B 0,C 180,E1 -25769.4,E2 -25769.4} C_VEL
LIN {X 0,Y 156.98,Z 195.295,A -85,B 0,C 180,E1 -25772.591,E2 -25772.591} C_VEL
LIN {X 0,Y 161.928,Z 204.104,A -85,B 0,C 180,E1 -25776.287,E2 -25776.287} C_VEL
LIN {X 0,Y 166.26,Z 212.962,A -85,B 0,C 180,E1 -25779.169,E2 -25779.169} C_VEL
LIN {X 0,Y 167.24,Z 215.497,A -85,B 0,C 180,E1 -25779.812,E2 -25779.812} C_VEL
LIN {X 0,Y 162.803,Z 267.324,A -85,B 0,C 180,E1 -25781.567,E2 -25781.567} C_VEL
LIN {X 0,Y 160.66,Z 281.341,A -85,B 0,C 180,E1 -25782.423,E2 -25782.423} C_VEL
LIN {X 0,Y 157.403,Z 295.766,A -85,B 0,C 180,E1 -25783.717,E2 -25783.717} C_VEL
LIN {X 0,Y 153.583,Z 308.565,A -85,B 0,C 180,E1 -25785.287,E2 -25785.287} C_VEL
LIN {X 0,Y 149.014,Z 321.009,A -85,B 0,C 180,E1 -25787.315,E2 -25787.315} C_VEL
LIN {X 0,Y 143.676,Z 333.522,A -85,B 0,C 180,E1 -25790.058,E2 -25790.058} C_VEL
LIN {X 0,Y 139.062,Z 342.797,A -85,B 0,C 180,E1 -25792.667,E2 -25792.667} C_VEL
LIN {X 0,Y 133.369,Z 353.175,A -85,B 0,C 180,E1 -25796.407,E2 -25796.407} C_VEL
LIN {X 0,Y 128.218,Z 361.742,A -85,B 0,C 180,E1 -25800.442,E2 -25800.442} C_VEL
LIN {X 0,Y 123.167,Z 369.951,A -85,B 0,C 180,E1 -25805.564,E2 -25805.564} C_VEL
LIN {X 0,Y 118.95,Z 376.554,A -85,B 0,C 180,E1 -25811.036,E2 -25811.036} C_VEL
LIN {X 0,Y 115.549,Z 382.086,A -85,B 0,C 180,E1 -25817.223,E2 -25817.223} C_VEL
LIN {X 0,Y 113.585,Z 385.823,A -85,B 0,C 180,E1 -25822.892,E2 -25822.892} C_VEL
LIN {X 0,Y 112.338,Z 389.055,A -85,B 0,C 180,E1 -25830.001,E2 -25830.001} C_VEL
LIN {X 0,Y 112.092,Z 390.151,A -85,B 0,C 180,E1 -25833.595,E2 -25833.595} C_VEL
LIN {X 0,Y 112.125,Z 391.356,A -85,B 0,C 180,E1 -25840.839,E2 -25840.839} C_VEL
LIN {X 0,Y 113.38,Z 391.236,A -85,B 0,C 180,E1 -25848.056,E2 -25848.056} C_VEL
LIN {X 0,Y 116.106,Z 389.774,A -85,B 0,C 180,E1 -25855.07,E2 -25855.07} C_VEL
LIN {X 0,Y 120.174,Z 386.933,A -85,B 0,C 180,E1 -25861.759,E2 -25861.759} C_VEL
LIN {X 0,Y 125.664,Z 382.624,A -85,B 0,C 180,E1 -25867.967,E2 -25867.967} C_VEL
LIN {X 0,Y 132.492,Z 376.71,A -85,B 0,C 180,E1 -25873.598,E2 -25873.598} C_VEL
LIN {X 0,Y 139.367,Z 370.006,A -85,B 0,C 180,E1 -25878.058,E2 -25878.058} C_VEL
LIN {X 0,Y 146.913,Z 361.619,A -85,B 0,C 180,E1 -25882.123,E2 -25882.123} C_VEL
LIN {X 0,Y 153.966,Z 352.846,A -85,B 0,C 180,E1 -25885.249,E2 -25885.249} C_VEL
LIN {X 0,Y 160.223,Z 344.156,A -85,B 0,C 180,E1 -25887.606,E2 -25887.606} C_VEL
LIN {X 0,Y 167.067,Z 332.929,A -85,B 0,C 180,E1 -25890.004,E2 -25890.004} C_VEL
LIN {X 0,Y 172.654,Z 322.446,A -85,B 0,C 180,E1 -25891.674,E2 -25891.674} C_VEL
LIN {X 0,Y 178.116,Z 310.059,A -85,B 0,C 180,E1 -25893.218,E2 -25893.218} C_VEL
LIN {X 0,Y 182.993,Z 296.228,A -85,B 0,C 180,E1 -25894.494,E2 -25894.494} C_VEL
LIN {X 0,Y 186.653,Z 282.233,A -85,B 0,C 180,E1 -25895.458,E2 -25895.458} C_VEL
LIN {X 0,Y 189.292,Z 267.91,A -85,B 0,C 180,E1 -25896.091,E2 -25896.091} C_VEL
LIN {X 0,Y 192.381,Z 236.184,A -85,B 0,C 180,E1 -25897.017,E2 -25897.017} C_VEL
LIN {X 0,Y 188.579,Z 228.193,A -85,B 0,C 180,E1 -25900.26,E2 -25900.26} C_VEL
LIN {X 0,Y 184.861,Z 221.186,A -85,B 0,C 180,E1 -25904,E2 -25904} C_VEL
LIN {X 0,Y 182.583,Z 217.289,A -85,B 0,C 180,E1 -25906.735,E2 -25906.735} C_VEL
LIN {X 0,Y 180.626,Z 213.793,A -85,B 0,C 180,E1 -25909.614,E2 -25909.614} C_VEL
LIN {X 0,Y 178.608,Z 210.07,A -85,B 0,C 180,E1 -25913.575,E2 -25913.575} C_VEL
LIN {X 0,Y 176.864,Z 206.499,A -85,B 0,C 180,E1 -25920.321,E2 -25920.321} C_VEL
LIN {X 0,Y 176.843,Z 205.789,A -85,B 0,C 180,E1 -25921.287,E2 -25921.287} C_VEL
LIN {X 0,Y 176.84,Z 206.025,A -85,B 0,C 180,E1 -25924.714,E2 -25924.714} C_VEL
LIN {X 0,Y 177.969,Z 209.608,A -85,B 0,C 180,E1 -25930.674,E2 -25930.674} C_VEL
LIN {X 0,Y 178.925,Z 210.757,A -85,B 0,C 180,E1 -25932.908,E2 -25932.908} C_VEL
LIN {X 0,Y 181.397,Z 215.184,A -85,B 0,C 180,E1 -25937.328,E2 -25937.328} C_VEL
LIN {X 0,Y 183.786,Z 219.333,A -85,B 0,C 180,E1 -25940.495,E2 -25940.495} C_VEL
LIN {X 0,Y 185.466,Z 222.776,A -85,B 0,C 180,E1 -25942.445,E2 -25942.445} C_VEL
LIN {X 0,Y 188.112,Z 229.17,A -85,B 0,C 180,E1 -25945.222,E2 -25945.222} C_VEL
LIN {X 0,Y 191.247,Z 237.509,A -85,B 0,C 180,E1 -25948.12,E2 -25948.12} C_VEL
LIN {X 0,Y 192.067,Z 239.922,A -85,B 0,C 180,E1 -25948.832,E2 -25948.832} C_VEL
LIN {X 0,Y 189.073,Z 271.191,A -85,B 0,C 180,E1 -25949.745,E2 -25949.745} C_VEL
LIN {X 0,Y 186.329,Z 286.024,A -85,B 0,C 180,E1 -25950.367,E2 -25950.367} C_VEL
LIN {X 0,Y 182.415,Z 300.387,A -85,B 0,C 180,E1 -25951.258,E2 -25951.258} C_VEL
LIN {X 0,Y 177.856,Z 313.137,A -85,B 0,C 180,E1 -25952.367,E2 -25952.367} C_VEL
LIN {X 0,Y 172.352,Z 325.565,A -85,B 0,C 180,E1 -25953.815,E2 -25953.815} C_VEL
LIN {X 0,Y 165.657,Z 338.101,A -85,B 0,C 180,E1 -25955.769,E2 -25955.769} C_VEL
LIN {X 0,Y 158.623,Z 349.29,A -85,B 0,C 180,E1 -25958.147,E2 -25958.147} C_VEL
LIN {X 0,Y 151.345,Z 359.321,A -85,B 0,C 180,E1 -25961.009,E2 -25961.009} C_VEL
LIN {X 0,Y 144.407,Z 367.672,A -85,B 0,C 180,E1 -25964.122,E2 -25964.122} C_VEL
LIN {X 0,Y 137.948,Z 374.655,A -85,B 0,C 180,E1 -25967.542,E2 -25967.542} C_VEL
LIN {X 0,Y 131.158,Z 381.316,A -85,B 0,C 180,E1 -25971.959,E2 -25971.959} C_VEL
LIN {X 0,Y 124.431,Z 387.248,A -85,B 0,C 180,E1 -25977.551,E2 -25977.551} C_VEL
LIN {X 0,Y 120.425,Z 390.691,A -85,B 0,C 180,E1 -25982.167,E2 -25982.167} C_VEL
LIN {X 0,Y 116.144,Z 394.001,A -85,B 0,C 180,E1 -25988.711,E2 -25988.711} C_VEL
LIN {X 0,Y 113.428,Z 395.937,A -85,B 0,C 180,E1 -25995.65,E2 -25995.65} C_VEL
LIN {X 0,Y 112.239,Z 396.552,A -85,B 0,C 180,E1 -26002.805,E2 -26002.805} C_VEL
LIN {X 0,Y 112.105,Z 396.126,A -85,B 0,C 180,E1 -26008.055,E2 -26008.055} C_VEL
LIN {X 0,Y 112.202,Z 395.844,A -85,B 0,C 180,E1 -26009.999,E2 -26009.999} C_VEL
LIN {X 0,Y 112.107,Z 394.972,A -85,B 0,C 180,E1 -26013.594,E2 -26013.594} C_VEL
LIN {X 0,Y 112.597,Z 392.178,A -85,B 0,C 180,E1 -26020.792,E2 -26020.792} C_VEL
LIN {X 0,Y 113.015,Z 390.898,A -85,B 0,C 180,E1 -26023.155,E2 -26023.155} C_VEL
LIN {X 0,Y 113.102,Z 389.256,A -85,B 0,C 180,E1 -26026.028,E2 -26026.028} C_VEL
LIN {X 0,Y 111.984,Z 386.092,A -85,B 0,C 180,E1 -26030.784,E2 -26030.784} C_VEL
LIN {X 0,Y 111.45,Z 382.357,A -85,B 0,C 180,E1 -26035.508,E2 -26035.508} C_VEL
LIN {X 0,Y 112.428,Z 379.759,A -85,B 0,C 180,E1 -26038.193,E2 -26038.193} C_VEL
LIN {X 0,Y 116.944,Z 372.88,A -85,B 0,C 180,E1 -26043.772,E2 -26043.772} C_VEL
LIN {X 0,Y 122.711,Z 364.091,A -85,B 0,C 180,E1 -26049.049,E2 -26049.049} C_VEL
LIN {X 0,Y 128.464,Z 354.896,A -85,B 0,C 180,E1 -26053.144,E2 -26053.144} C_VEL
LIN {X 0,Y 134.813,Z 343.734,A -85,B 0,C 180,E1 -26056.872,E2 -26056.872} C_VEL
LIN {X 0,Y 140.395,Z 332.303,A -85,B 0,C 180,E1 -26059.764,E2 -26059.764} C_VEL
LIN {X 0,Y 145.184,Z 321.255,A -85,B 0,C 180,E1 -26061.87,E2 -26061.87} C_VEL
LIN {X 0,Y 149.537,Z 309.402,A -85,B 0,C 180,E1 -26063.595,E2 -26063.595} C_VEL
LIN {X 0,Y 153.395,Z 296.499,A -85,B 0,C 180,E1 -26064.981,E2 -26064.981} C_VEL
LIN {X 0,Y 156.522,Z 282.24,A -85,B 0,C 180,E1 -26066.093,E2 -26066.093} C_VEL
LIN {X 0,Y 158.589,Z 268.816,A -85,B 0,C 180,E1 -26066.744,E2 -26066.744} C_VEL
LIN {X 0,Y 162.62,Z 221.082,A -85,B 0,C 180,E1 -26068.399,E2 -26068.399} C_VEL
LIN {X 0,Y 158.754,Z 210.074,A -85,B 0,C 180,E1 -26071.392,E2 -26071.392} C_VEL
LIN {X 0,Y 156.688,Z 205.109,A -85,B 0,C 180,E1 -26073.081,E2 -26073.081} C_VEL
LIN {X 0,Y 153.092,Z 198.785,A -85,B 0,C 180,E1 -26076.137,E2 -26076.137} C_VEL
LIN {X 0,Y 149.992,Z 193.558,A -85,B 0,C 180,E1 -26079.167,E2 -26079.167} C_VEL
LIN {X 0,Y 147.038,Z 189.085,A -85,B 0,C 180,E1 -26082.513,E2 -26082.513} C_VEL
LIN {X 0,Y 144.706,Z 185.425,A -85,B 0,C 180,E1 -26085.711,E2 -26085.711} C_VEL
LIN {X 0,Y 142.365,Z 181.992,A -85,B 0,C 180,E1 -26089.731,E2 -26089.731} C_VEL
LIN {X 0,Y 142,Z 181.017,A -85,B 0,C 180,E1 -26090.584,E2 -26090.584} C_VEL
LIN {X 0,Y 139.469,Z 177.589,A -85,B 0,C 180,E1 -26098.557,E2 -26098.557} C_VEL
LIN {X 0,Y 139.312,Z 175.896,A -85,B 0,C 180,E1 -26101.168,E2 -26101.168} C_VEL
LIN {X 0,Y 139.223,Z 176.152,A -85,B 0,C 180,E1 -26104.343,E2 -26104.343} C_VEL
LIN {X 0,Y 140.971,Z 180.413,A -85,B 0,C 180,E1 -26113.58,E2 -26113.58} C_VEL
LIN {X 0,Y 142.065,Z 181.428,A -85,B 0,C 180,E1 -26115.998,E2 -26115.998} C_VEL
LIN {X 0,Y 144.068,Z 184.84,A -85,B 0,C 180,E1 -26119.735,E2 -26119.735} C_VEL
LIN {X 0,Y 145.198,Z 186.239,A -85,B 0,C 180,E1 -26121.398,E2 -26121.398} C_VEL
LIN {X 0,Y 148.207,Z 190.89,A -85,B 0,C 180,E1 -26125.264,E2 -26125.264} C_VEL
LIN {X 0,Y 151.07,Z 195.471,A -85,B 0,C 180,E1 -26128.325,E2 -26128.325} C_VEL
LIN {X 0,Y 154.637,Z 201.525,A -85,B 0,C 180,E1 -26131.608,E2 -26131.608} C_VEL
LIN {X 0,Y 159.144,Z 209.953,A -85,B 0,C 180,E1 -26135.201,E2 -26135.201} C_VEL
LIN {X 0,Y 162.835,Z 217.868,A -85,B 0,C 180,E1 -26137.842,E2 -26137.842} C_VEL
LIN {X 0,Y 158.521,Z 267.309,A -85,B 0,C 180,E1 -26139.549,E2 -26139.549} C_VEL
LIN {X 0,Y 156.315,Z 281.337,A -85,B 0,C 180,E1 -26140.402,E2 -26140.402} C_VEL
LIN {X 0,Y 153.233,Z 294.684,A -85,B 0,C 180,E1 -26141.569,E2 -26141.569} C_VEL
LIN {X 0,Y 149.268,Z 307.752,A -85,B 0,C 180,E1 -26143.132,E2 -26143.132} C_VEL
LIN {X 0,Y 144.479,Z 320.388,A -85,B 0,C 180,E1 -26145.144,E2 -26145.144} C_VEL
LIN {X 0,Y 139.406,Z 331.877,A -85,B 0,C 180,E1 -26147.602,E2 -26147.602} C_VEL
LIN {X 0,Y 134.564,Z 341.452,A -85,B 0,C 180,E1 -26150.225,E2 -26150.225} C_VEL
LIN {X 0,Y 128.471,Z 352.084,A -85,B 0,C 180,E1 -26153.98,E2 -26153.98} C_VEL
LIN {X 0,Y 122.969,Z 360.86,A -85,B 0,C 180,E1 -26158.086,E2 -26158.086} C_VEL
LIN {X 0,Y 117.482,Z 369.267,A -85,B 0,C 180,E1 -26163.343,E2 -26163.343} C_VEL
LIN {X 0,Y 113.463,Z 375.147,A -85,B 0,C 180,E1 -26168.184,E2 -26168.184} C_VEL
LIN {X 0,Y 109.191,Z 381.434,A -85,B 0,C 180,E1 -26175.081,E2 -26175.081} C_VEL
LIN {X 0,Y 106.547,Z 386.1,A -85,B 0,C 180,E1 -26182.42,E2 -26182.42} C_VEL
LIN {X 0,Y 105.233,Z 389.282,A -85,B 0,C 180,E1 -26190.001,E2 -26190.001} C_VEL
LIN {X 0,Y 104.968,Z 390.36,A -85,B 0,C 180,E1 -26193.84,E2 -26193.84} C_VEL
LIN {X 0,Y 105.085,Z 391.529,A -85,B 0,C 180,E1 -26201.575,E2 -26201.575} C_VEL
LIN {X 0,Y 106.567,Z 391.374,A -85,B 0,C 180,E1 -26209.254,E2 -26209.254} C_VEL
LIN {X 0,Y 109.606,Z 389.876,A -85,B 0,C 180,E1 -26216.67,E2 -26216.67} C_VEL
LIN {X 0,Y 114.072,Z 386.997,A -85,B 0,C 180,E1 -26223.676,E2 -26223.676} C_VEL
LIN {X 0,Y 120.045,Z 382.649,A -85,B 0,C 180,E1 -26230.091,E2 -26230.091} C_VEL
LIN {X 0,Y 127.35,Z 376.685,A -85,B 0,C 180,E1 -26235.843,E2 -26235.843} C_VEL
LIN {X 0,Y 134.633,Z 369.922,A -85,B 0,C 180,E1 -26240.351,E2 -26240.351} C_VEL
LIN {X 0,Y 141.416,Z 362.827,A -85,B 0,C 180,E1 -26243.861,E2 -26243.861} C_VEL
LIN {X 0,Y 148.711,Z 354.271,A -85,B 0,C 180,E1 -26247.02,E2 -26247.02} C_VEL
LIN {X 0,Y 156.399,Z 344.019,A -85,B 0,C 180,E1 -26249.796,E2 -26249.796} C_VEL
